(* CODESYS project PLC 1 Simulatie Ladder StructuredTekst IOStructures 2V0.project
   Title: Simulatie Sorteer Station
   Author: Rene Potters/Gerard Harkema
   Version: 0.1.0
   Description: Simulatie voor opstelling Sorteer Station.
   Company: Avans

Project tree, tasks and I/O mapping:
  Device : EHV-CPU1025, Hitachi-IES, order no. EHV-CPU1025, version 3.5.4.11
      settings: IP Address = '192.168.1.31'
    application ApplicationLadder
      libraries: VisuDialogs, * (System); Standard, 3.5.14.0 (System); Util, 3.5.14.0 (System)
      task MainTask (cyclic, interval t#20ms, priority 1) calls BedieningPrg, HoofdPrg, MagazijnPrg, OverzetterPrg, SorterenPrg, SignaleringPrg
      task Simulatie (cyclic, interval 50 ms, priority 1) calls MagazijnSim [Afhandeling Magazijn], OverzetterSim [Afhandeling Overzetter], SorterenSim [Afhandeling Sorteren]
    application ApplicationSt
      libraries: Standard, * (System); Util, * (System); VisuDialogs, 3.5.12.0 (System)
      task MainTask (cyclic, interval t#20ms, priority 1) calls Main
      task Simulatie (cyclic, interval t#20ms, priority 1) calls MagazijnSim, OverzetterSim, SorterenSim
    application MagazijnTest
      libraries: Standard, * (System); Util, * (System); VisuDialogs, 3.5.12.0 (System)
      task MainTask (cyclic, interval t#20ms, priority 1) calls MagazijnTest
      task Simulatie (cyclic, interval t#20ms, priority 1) calls MagazijnSim
    application OverzetterTest
      libraries: Standard, * (System); Util, * (System); VisuDialogs, 3.5.12.0 (System)
      task MainTask (cyclic, interval t#20ms, priority 1) calls OverzetterTest
      task Simulatie (cyclic, interval t#20ms, priority 1) calls OverzetterSim
    application SorteerTest
      libraries: Standard, * (System); Util, * (System); VisuDialogs, 3.5.12.0 (System)
      task MainTask (cyclic, interval t#20ms, priority 1) calls SorteerTest
      task Simulatie (cyclic, interval 20 ms, priority 1) calls SorterenSim
    application UitvoerGootTest
      libraries: Standard, * (System); Util, * (System); VisuDialogs, 3.5.12.0 (System)
      task MainTask (cyclic, interval t#20ms, priority 1) calls UitvoerGootTest
      task Simulatie (cyclic, interval t#20ms, priority 1) calls SorterenSim
    Basic : Basic, Hitachi-IES, version 3.4.4.0
      <Empty>
      <Empty>
      <Empty>
      <Empty>
      <Empty>
      <Empty>
      <Empty>
      <Empty>
      <Empty>
      <Empty>
      <Empty>
  Simulatie/
    program MagazijnSim [ST]
    program SorterenSim [ST]
    global variables SIM
    program OverzetterSim [ST]
    data type OverzetterDUT
    data type SorterenDUT
    data type MagazijnDUT
    function block SorterenGootSim [ST]
  Programma Ladder/
    program MagazijnPrg [SFC]
    program HoofdPrg [SFC]
    program OverzetterPrg [SFC]
    program SorterenPrg [SFC]
    program BedieningPrg [LD]
    program SignaleringPrg [LD]
  text list GlobalTextList
  Programma Structured Text/
    function block OverzetterClass [ST]: initialize, cycle, isError, isKlaar, reset, start, noodstop
    function block SorteerGootClass [ST]: initialize, cycle, isError, isKlaar, start, reset, noodstop, isGootVol, productTellerReset
    function block MagazijnClass [ST]: initialize, cycle, start, isMagazijnLeeg, isError, reset, isKlaar, noodstop
    program Main [ST]
    function block SorteerStationClass [ST]: initialize, cycle
    TestProgramms/
      program MagazijnTest [ST]
      program OverzetterTest [ST]
      program SorteerTest [ST]
      program UitvoerGootTest [ST]
    States/
      data type magazijnStates
      data type overzetterStates
      data type sorteerStationStates
      data type sorteerStates
      data type uitvoerGootStates
    function block MeetstationClass [ST]: initialize, getProductType
    data type productType
    function block UitvoerGootClass [ST]: cycle, initialize, isError, noodstop, reset, gaUit, gaIn, isUit, isIn
    Structures/
      data type uitvoerGootIO
      data type sorteerGootIO
      data type meetstationIO
      data type magazijnIO
      data type overzetterIO
      data type sorteerStationIO
      data type hmiIO
  global variables GVL
  Visualisaties/
    visualisation SorteerStationHMI
    visualisation BekerMagazijnHMI
    visualisation OverzetterHMI
    visualisation SorterenHMI
*)

// Simulatie/OverzetterDUT
{attribute 'qualified_only'}
{attribute 'strict'}
TYPE OverzetterDUT :
(
	INHETMIDDEN, NAARRECHTS, ISRECHTS, NAARLINKS, ISLINKS, GEVALLEN
);
END_TYPE

// Simulatie/SorterenDUT
{attribute 'qualified_only'}
{attribute 'strict'}
TYPE SorterenDUT :
(
	VOLGENDEBLOK, OPDEBAND, VOORSTOPPER, NAARGOOT1, INGOOT1, NAARGOOT2, INGOOT2, NAARGOOT3, INGOOT3, GEREED, VOL
);
END_TYPE

// Simulatie/MagazijnDUT
{attribute 'qualified_only'}
{attribute 'strict'}
TYPE MagazijnDUT :
(
	INGETROKKEN, INTREKKEN, UITGESTOTEN, UITSTOTEN, LEEG
);
END_TYPE

// Programma Structured Text/States/magazijnStates
// Datum : 17 december 2020, Auteur: Gerard Harkema
{attribute 'qualified_only'}
{attribute 'strict'}
TYPE magazijnStates :
(
	idle := 0,
	in,
	travel_out,
	out,
	travel_in,
	error
);
END_TYPE

// Programma Structured Text/States/overzetterStates
// Datum : 17 december 2020, Auteur: Gerard Harkema
{attribute 'qualified_only'}
{attribute 'strict'}
TYPE overzetterStates :
(
	idle := 0,
	is_links,
	vaccuum_aanzetten,
	ga_naar_rechts,
	is_rechts,
	vaccuum_lossen,
	ga_naar_midden,
	is_midden,
	ga_naar_links,
	error
);
END_TYPE

// Programma Structured Text/States/sorteerStationStates
// Datum : 17 december 2020, Auteur: Gerard Harkema
{attribute 'qualified_only'}
{attribute 'strict'}
TYPE sorteerStationStates :
(
	idle := 0,
	wacht_op_klaar,
	wacht_enable,
	product_uitgifte,
	product_overzetten,
	product_sorteren,
	service,
	error
);
END_TYPE

// Programma Structured Text/productType
// Datum : 17 december 2020, Auteur: Gerard Harkema
{attribute 'qualified_only'}
{attribute 'strict'}
TYPE productType :
(
	onbekend := 0,
	metaal_blank,
	metaal_zwart,
	kunstof_rood,
	kunstof_zwart
);
END_TYPE

// Programma Structured Text/States/sorteerStates
// Datum : 17 december 2020, Auteur: Gerard Harkema
{attribute 'qualified_only'}
{attribute 'strict'}
TYPE sorteerStates :
(
	idle := 0,
	wacht_op_start,
	stopper_uit,
	meten,
	uitvoer_goot_uit,
	transporteren_naar_goot,
	uitvoer_goot_in,
	goot_vol,
	error,
	reset_error
);
END_TYPE

// Programma Structured Text/States/uitvoerGootStates
// Datum : 17 december 2020, Auteur: Gerard Harkema
{attribute 'qualified_only'}
{attribute 'strict'}
TYPE uitvoerGootStates :
(
	idle := 0,
	is_in,
	ga_in,
	is_uit,
	ga_uit,
	error
);
END_TYPE

// Programma Structured Text/Structures/uitvoerGootIO
// Datum : 17 december 2020, Auteur: Gerard Harkema
TYPE uitvoerGootIO :
STRUCT
	//Pusher uitvoergoo is in
	Ix_UitvoerGootIsIn 		: REFERENCE TO BOOL;
	//Pusher uitvoergoot is uit
	Ix_UitvoerGootIsUit 	: REFERENCE TO BOOL;
	//Pusher goot uit
	Qx_UitvoerGootUit 		: REFERENCE TO BOOL;
END_STRUCT
END_TYPE

// Programma Structured Text/Structures/sorteerGootIO
// Datum : 17 december 2020, Auteur: Gerard Harkema
TYPE sorteerGootIO :
STRUCT
		//Product is naar een van de goten gegaan
	Ix_BekerInGoot 			:REFERENCE TO BOOL;
	//Pusher uitvoergoot 1 is in
	Ix_UitvoerGoot1IsIn 	:REFERENCE TO BOOL;
	//Pusher uitvoergoot 2 is in
	Ix_UitvoerGoot2IsIn 	:REFERENCE TO BOOL;
	//Beker afvoeren is bezig
	Ix_StationAfvoerVrij 	:REFERENCE TO BOOL;
	//Pusher uitvoergoot 1 is uit
	Ix_UitvoerGoot1IsUit 	:REFERENCE TO BOOL;
	//Pusher uitvoergoot 2 is uit
	Ix_UitvoerGoot2IsUit 	:REFERENCE TO BOOL;

	//Transportband aan
	Qx_MotorAfvoerAan 		:REFERENCE TO BOOL;
	//Pusher goot 1 uit
	Qx_UitvoerGoot1Uit 		:REFERENCE TO BOOL;
	//Pusher goot 2 uit
	Qx_UitvoerGoot2Uit 		:REFERENCE TO BOOL;
	//Beker stoppen op band voor detectie
	Qx_StopperUit 			:REFERENCE TO BOOL;
	//Uitsorteren is bezet
	Qx_StationBezet 		:REFERENCE TO BOOL;
	
	uitvoerGoot1			:uitvoerGootIO;
	uitvoerGoot2			:uitvoerGootIO;
	meetstation				:meetstationIO;

 
END_STRUCT
END_TYPE

// Programma Structured Text/Structures/meetstationIO
// Datum : 17 december 2020, Auteur: Gerard Harkema
TYPE meetstationIO :
STRUCT
	//Beker aanwezig op detectiepositie
	Ix_BekerAanwezig :REFERENCE TO BOOL;
	//Beker is van aluminium
	Ix_BekerMetaal :REFERENCE TO BOOL;
	//Beker reflecteert en is dus niet zwart
	Ix_BekerReflecteerd :REFERENCE TO BOOL;
END_STRUCT
END_TYPE

// Programma Structured Text/Structures/magazijnIO
// Datum : 17 december 2020, Auteur: Gerard Harkema
TYPE magazijnIO :
STRUCT
	// Bekers magazijn zijn op
	Ix_MagazijnLeeg				: REFERENCE TO BOOL;
	// Beker is uit dekselmagazijn gestoten
	Ix_UitstoterBekerIn			: REFERENCE TO BOOL;
	// Uitstoter Beker haalt nieuwe beker op
	Ix_UitstoterBekerUit		: REFERENCE TO BOOL;
	// Beker uit magazijn stoten
	Qx_BekerUitstoten			: REFERENCE TO BOOL;

	//Perslucht is aanwezig
	Ix_PersluchtAanwezig 		: REFERENCE TO BOOL;

END_STRUCT
END_TYPE

// Programma Structured Text/Structures/overzetterIO
// Datum : 17 december 2020, Auteur: Gerard Harkema
TYPE overzetterIO :
STRUCT
	//Werkstuk door overzetter opgepakt
	Ix_VacuumAanwezig 		:REFERENCE TO BOOL;
	//Overzetter haalt beker op(linker pos.)
	Ix_OverzetterIsLinks 	:REFERENCE TO BOOL;
	//Overzetter plaatst beker op sorteerpositie
	Ix_OverzetterIsRechts 	:REFERENCE TO BOOL;
	//Beker aanwezig op detectiepositie
	
		//Beker oppakken
	Qx_VacuumAan 			:REFERENCE TO BOOL;
	//Beker loslaten
	Qx_BekerLossen 			:REFERENCE TO BOOL;
	//Overzetter naar bekermagazijn
	Qx_OverzetterLinks 		:REFERENCE TO BOOL;
	//Overzetter naar sorteerpositie
	Qx_OverzetterRechts 	:REFERENCE TO BOOL;

END_STRUCT
END_TYPE

// Programma Structured Text/Structures/sorteerStationIO
// Datum : 17 december 2020, Auteur: Gerard Harkema
TYPE sorteerStationIO :
STRUCT
	magazijn		: magazijnIO;
	overzetter		: overzetterIO;
	sorteerGoot		: sorteerGootIO;
	hmi				: hmiIO;
END_STRUCT
END_TYPE

// Programma Structured Text/Structures/hmiIO
// Datum : 17 december 2020, Auteur: Gerard Harkema
TYPE hmiIO :
STRUCT
	// Indrukken resetknop 
	Ix_Resetknop			: REFERENCE TO BOOL;
	// Keuzeknop staat op hand
	Ix_Hand					: REFERENCE TO BOOL;
	// Keuzeknop staat op auto
	Ix_Auto					: REFERENCE TO BOOL;
	// Indrukken noodstop
	Ix_Noodstop				: REFERENCE TO BOOL;
	// Bekers magazijn zijn op

	// Indrukken startknop
	Ix_Stopknop				: REFERENCE TO BOOL;
	// Indrukken stopknop
	Ix_Startknop			: REFERENCE TO BOOL;	
	//Perslucht is aanwezig

	// Visualisatie invisible Gele vlak
	Qx_GeleLamp				: REFERENCE TO BOOL;
	// Visualisatie invisible groene vlak
	Qx_GroeneLamp			: REFERENCE TO BOOL;
	// Visualisatie invisible rode vlak
	Qx_RodeLamp				: REFERENCE TO BOOL;

END_STRUCT
END_TYPE

// Simulatie/SIM
{attribute 'qualified_only'}
VAR_GLOBAL
	// Rotatie van de overzetter
	Vx_OvzRotate: INT := 0;
	// Visualisatie invisible blok
	Vx_OvzBlokLinks: BOOL := FALSE;
	// Visualisatie invisible blok
	Vx_OvzBlokOverzetter: BOOL := FALSE;
	// Visualisatie invisible blok
	Vx_OvzBlokRechts: BOOL := FALSE;
	// Visualisatie invisible blok
	Vx_OvzBlokGevallen: BOOL := FALSE;	
	// Magazijn opnieuw vullen (simulatie)
	Ix_MagazijnVullen 	: BOOL;
	// Goten legen (symulatie)
	Ix_GotenLegen	  	: BOOL;
	
	
	
	
	
	
	
	
	
	
	
	
	
	
	
	
	
	
	
	
	
	
	
	
	
	
	
	
	
	
	
	
	
	
	
	
	
	
	
	
	
	
	
	
	
	
	
	
	// Simulatie visualisatie 
	Vw_Rotate45: INT := 45;
	// Visualisatie X positie van de uitstoter
	Vw_MagUitstoterBekerX: INT := 30;
	// Visualisatie invisible blok uitgestoten
	Vx_MagBlokUit: BOOL := TRUE;
	// Visualisatie invisible blok 1
	Vx_MagBlok1: BOOL := TRUE;
	// Visualisatie invisible blok 2
	Vx_MagBlok2: BOOL := TRUE;
	// Visualisatie invisible blok 3
	Vx_MagBlok3: BOOL := TRUE;
	// Visualisatie invisible blok 4
	Vx_MagBlok4: BOOL := TRUE;
	// Visualisatie invisible blokken
	Vx_MagBlok: ARRAY[1..8] OF BOOL;
	// Aantal blokken in het magazijn
	Vw_MagBlokAantal: INT := 4;
	// Simulatie onthoudt dat een blok maar 1x wordt uitgestoten
	Vw_MagBlok1X: INT := 0;
	// Ligt er een blok op band
	Vw_SorBlokBand: BOOL := FALSE;
	// Rotatie van de stopper
	Vw_SorStopperRotate: INT := 0;
	// Rotatie van de stopper goot 1
	Vw_SorGoot1Rotate: INT := 0;
	// Rotatie van de stopper goot 2
	Vw_SorGoot2Rotate: INT := 0;
	// Kleur van de blok op betreffende positie
	Vw_SorKleurBand: DWORD := 0;
	// Bewegen van de blok over de band
	Vi_SorBlokBandX: INT := 0;
	// Bewegen van de blok over de band
	Vi_SorBlokBandY: INT := 0;
	// Simulatie error. Inverse logica.
	Vx_MagLuchtDrukError: BOOL := TRUE;
	// Simulatie error. Inverse logica.
	Vx_MagIsInError: BOOL := TRUE;
	// Simulatie error. Inverse logica.
	Vx_MagIsUitError: BOOL := TRUE;
	// Simulatie error. Inverse logica.
	Vx_OvzLuchtDrukError: BOOL := TRUE;
	// Simulatie error. Inverse logica.
	Vx_OvzIsLinksError: BOOL := TRUE;
	// Simulatie error. Inverse logica.
	Vx_OvzIsRechtsError: BOOL := TRUE;
	// Simulatie error. Inverse logica.
	Vx_OvzVacuumError: BOOL := TRUE;
	// Simulatie error. Inverse logica.
	Vx_SorMotorAfvoerError: BOOL := TRUE;
	// Simulatie error. Inverse logica.
	Vx_SorGoot1InError: BOOL := TRUE;
	// Simulatie error. Inverse logica.
	Vx_SorGoot1UitError: BOOL := TRUE;
	// Simulatie error. Inverse logica.
	Vx_SorInGootError: BOOL := TRUE;
	// Ligt er een blok op de betreffende positie
	Vx_SorBlokGoot: ARRAY [1..3,1..6] OF BOOL;
	// Kleur van de blok op betreffende positie
	Vw_SorKleurGoot: ARRAY [1..3,1..6] OF DWORD;
END_VAR

// GVL
VAR_GLOBAL
	// Indrukken resetknop 
	Ix_Resetknop: BOOL;
	// Keuzeknop staat op hand
	Ix_Hand: BOOL;
	// Keuzeknop staat op auto
	Ix_Auto: BOOL;
	// Indrukken noodstop
	Ix_Noodstop: BOOL;
	// Bekers magazijn zijn op
	Ix_MagazijnLeeg: BOOL;
	// Beker is uit dekselmagazijn gestoten
	Ix_UitstoterBekerIn: BOOL;
	// Uitstoter Beker haalt nieuwe beker op
	Ix_UitstoterBekerUit: BOOL;
	// Indrukken startknop
	Ix_Stopknop: BOOL := TRUE;
	// Indrukken stopknop
	Ix_Startknop: BOOL;	
	//Perslucht is aanwezig
	Ix_PersluchtAanwezig :BOOL;
	//Werkstuk door overzetter opgepakt
	Ix_VacuumAanwezig :BOOL;
	//Overzetter haalt beker op(linker pos.)
	Ix_OverzetterIsLinks :BOOL;
	//Overzetter plaatst beker op sorteerpositie
	Ix_OverzetterIsRechts :BOOL;
	//Beker aanwezig op detectiepositie
	Ix_BekerAanwezig :BOOL;
	//Beker is van aluminium
	Ix_BekerMetaal :BOOL;
	//Beker reflecteert en is dus niet zwart
	Ix_BekerReflecteerd :BOOL;
	//Product is naar een van de goten gegaan
	Ix_BekerInGoot :BOOL;
	//Pusher uitvoergoot 1 is in
	Ix_UitvoerGoot1IsIn :BOOL;
	//Pusher uitvoergoot 2 is in
	Ix_UitvoerGoot2IsIn :BOOL;
	//Beker afvoeren is bezig
	Ix_StationAfvoerVrij :BOOL;
	//Pusher uitvoergoot 1 is uit
	Ix_UitvoerGoot1IsUit :BOOL;
	//Pusher uitvoergoot 2 is uit
	Ix_UitvoerGoot2IsUit :BOOL;
	// Beker uit magazijn stoten
	Qx_BekerUitstoten: BOOL;	
	//Beker oppakken
	Qx_VacuumAan :BOOL;
	//Beker loslaten
	Qx_BekerLossen :BOOL;
	//Overzetter naar bekermagazijn
	Qx_OverzetterLinks :BOOL;
	//Overzetter naar sorteerpositie
	Qx_OverzetterRechts :BOOL;
	//Transportband aan
	Qx_MotorAfvoerAan :BOOL;
	//Pusher goot 1 uit
	Qx_UitvoerGoot1Uit :BOOL;
	//Pusher goot 2 uit
	Qx_UitvoerGoot2Uit :BOOL;
	//Beker stoppen op band voor detectie
	Qx_StopperUit :BOOL;
	//Uitsorteren is bezet
	Qx_StationBezet :BOOL;
	// Visualisatie invisible Gele vlak
	Qx_GeleLamp: BOOL;
	// Visualisatie invisible groene vlak
	Qx_GroeneLamp: BOOL;
	// Visualisatie invisible rode vlak
	Qx_RodeLamp: BOOL;
	
END_VAR

// Programma Ladder/BedieningPrg
PROGRAM BedieningPrg
VAR
END_VAR

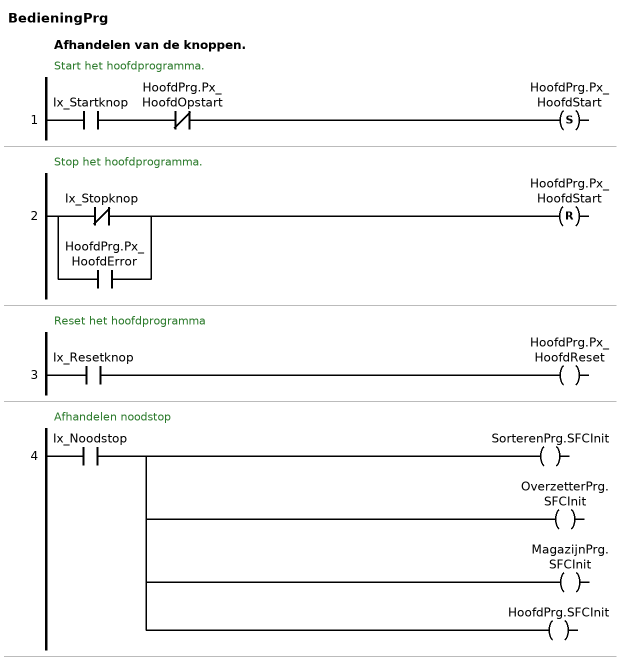
// NETWORK 1: Afhandelen van de knoppen.
// Start het hoofdprogramma.
HoofdPrg.Px_HoofdStart S= Ix_Startknop AND NOT HoofdPrg.Px_HoofdOpstart;

// NETWORK 2
// Stop het hoofdprogramma.
HoofdPrg.Px_HoofdStart R= NOT Ix_Stopknop OR HoofdPrg.Px_HoofdError;

// NETWORK 3
// Reset het hoofdprogramma
HoofdPrg.Px_HoofdReset := Ix_Resetknop;

// NETWORK 4
// Afhandelen noodstop
SorterenPrg.SFCInit := Ix_Noodstop;
OverzetterPrg.SFCInit := Ix_Noodstop;
MagazijnPrg.SFCInit := Ix_Noodstop;
HoofdPrg.SFCInit := Ix_Noodstop;

END_PROGRAM

// Programma Ladder/HoofdPrg
PROGRAM HoofdPrg
VAR_INPUT
	// Reset het programma
	Px_HoofdReset: BOOL;
	// Start het programma
	Px_HoofdStart: BOOL;
	// Reset de SFC bv Noodstop
	SFCInit: BOOL;
END_VAR
VAR_OUTPUT
	// Er is een error op getreden
	Px_HoofdError: BOOL;
	// Commando is uitgevoerd
	Px_HoofdGereed: BOOL;
	// Programma is bezig
	Px_HoofdBezig: BOOL;
	// Programma is aan het opstarten
	Px_HoofdOpstart: BOOL;
END_VAR

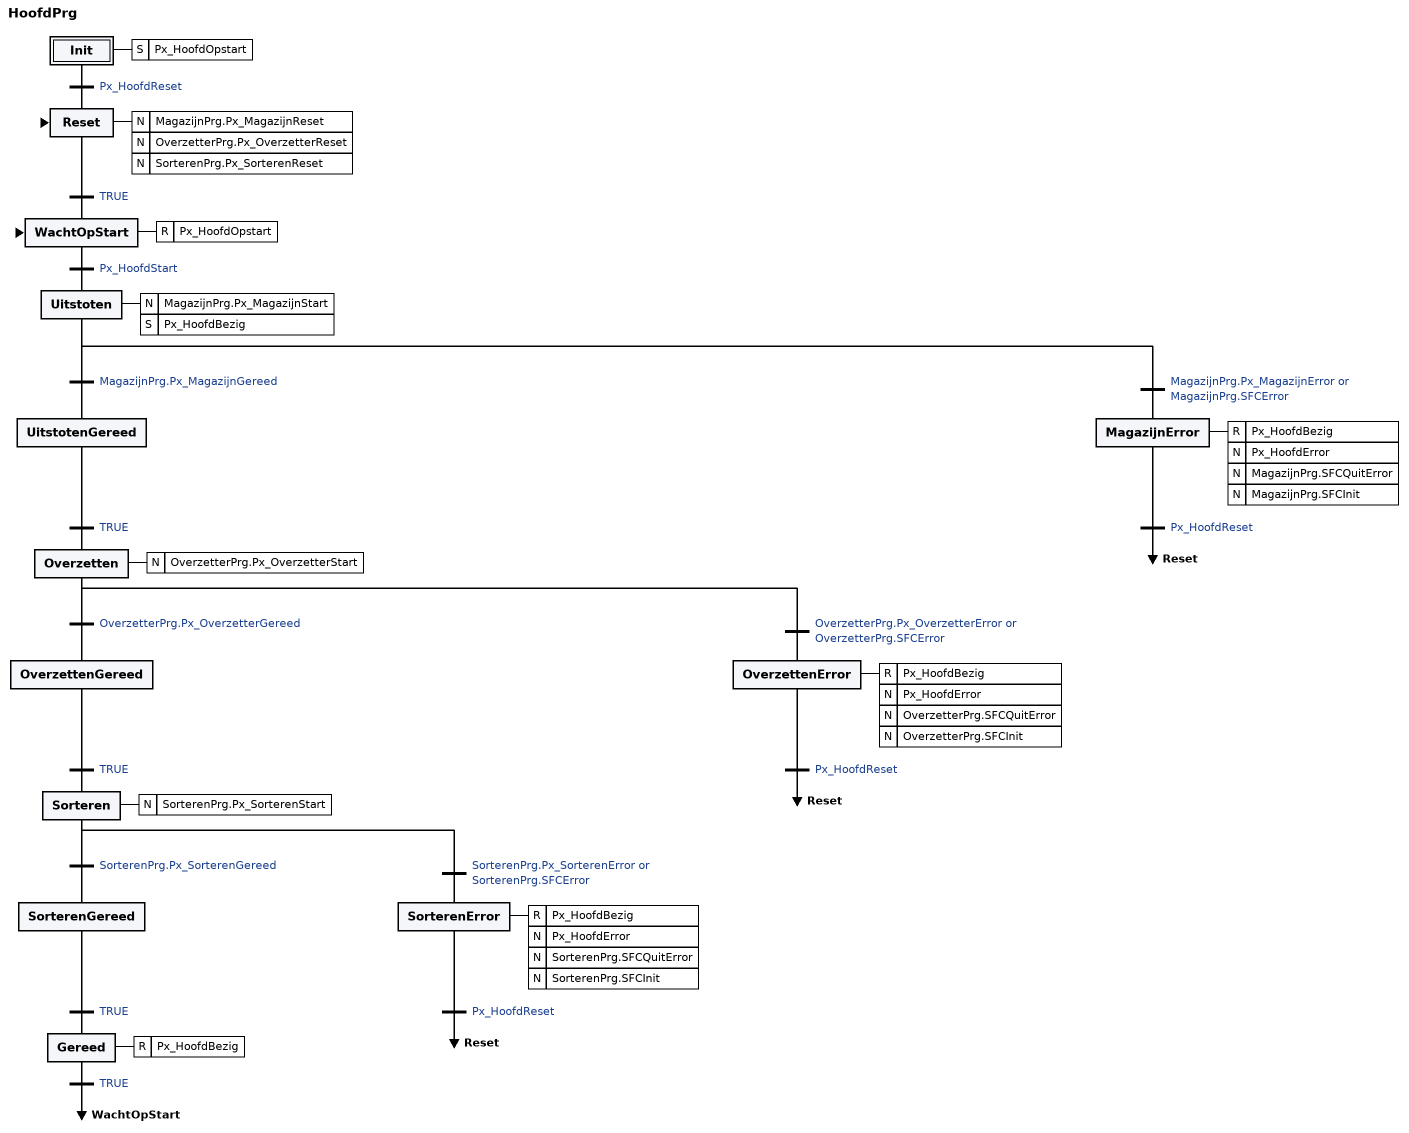
INITIAL_STEP Init:
    Px_HoofdOpstart(S);
END_STEP
TRANSITION FROM Init TO Reset
    := Px_HoofdReset;
END_TRANSITION
STEP Reset:
    MagazijnPrg.Px_MagazijnReset(N);
    OverzetterPrg.Px_OverzetterReset(N);
    SorterenPrg.Px_SorterenReset(N);
END_STEP
TRANSITION FROM Reset TO WachtOpStart
    := TRUE;
END_TRANSITION
STEP WachtOpStart:
    Px_HoofdOpstart(R);
END_STEP
TRANSITION FROM WachtOpStart TO Uitstoten
    := Px_HoofdStart;
END_TRANSITION
STEP Uitstoten:  // max time T#30S
    MagazijnPrg.Px_MagazijnStart(N);
    Px_HoofdBezig(S);
END_STEP
TRANSITION FROM Uitstoten TO UitstotenGereed
    := MagazijnPrg.Px_MagazijnGereed;
END_TRANSITION
STEP UitstotenGereed:
END_STEP
TRANSITION FROM UitstotenGereed TO Overzetten
    := TRUE;
END_TRANSITION
TRANSITION FROM Uitstoten TO MagazijnError
    := MagazijnPrg.Px_MagazijnError or MagazijnPrg.SFCError;
END_TRANSITION
STEP MagazijnError:
    Px_HoofdBezig(R);
    Px_HoofdError(N);
    MagazijnPrg.SFCQuitError(N);
    MagazijnPrg.SFCInit(N);
END_STEP
TRANSITION FROM MagazijnError TO Reset
    := Px_HoofdReset;
END_TRANSITION
STEP Overzetten:
    OverzetterPrg.Px_OverzetterStart(N);
END_STEP
TRANSITION FROM Overzetten TO OverzettenGereed
    := OverzetterPrg.Px_OverzetterGereed;
END_TRANSITION
STEP OverzettenGereed:
END_STEP
TRANSITION FROM OverzettenGereed TO Sorteren
    := TRUE;
END_TRANSITION
TRANSITION FROM Overzetten TO OverzettenError
    := OverzetterPrg.Px_OverzetterError or OverzetterPrg.SFCError;
END_TRANSITION
STEP OverzettenError:
    Px_HoofdBezig(R);
    Px_HoofdError(N);
    OverzetterPrg.SFCQuitError(N);
    OverzetterPrg.SFCInit(N);
END_STEP
TRANSITION FROM OverzettenError TO Reset
    := Px_HoofdReset;
END_TRANSITION
STEP Sorteren:
    SorterenPrg.Px_SorterenStart(N);
END_STEP
TRANSITION FROM Sorteren TO SorterenGereed
    := SorterenPrg.Px_SorterenGereed;
END_TRANSITION
STEP SorterenGereed:
END_STEP
TRANSITION FROM SorterenGereed TO Gereed
    := TRUE;
END_TRANSITION
TRANSITION FROM Sorteren TO SorterenError
    := SorterenPrg.Px_SorterenError or SorterenPrg.SFCError;
END_TRANSITION
STEP SorterenError:
    Px_HoofdBezig(R);
    Px_HoofdError(N);
    SorterenPrg.SFCQuitError(N);
    SorterenPrg.SFCInit(N);
END_STEP
TRANSITION FROM SorterenError TO Reset
    := Px_HoofdReset;
END_TRANSITION
STEP Gereed:
    Px_HoofdBezig(R);
END_STEP
TRANSITION FROM Gereed TO WachtOpStart
    := TRUE;
END_TRANSITION

END_PROGRAM

// Programma Ladder/SorterenPrg
PROGRAM SorterenPrg
VAR_INPUT
	// Reset de sorteren na start of error
	Px_SorterenReset: BOOL;
	// Start het sorteren
	Px_SorterenStart: BOOL;
	
	// Reset de SFC bv Noodstop
	SFCInit: BOOL;
	// Enable runtime limit checks
	SFCEnableLimit: BOOL := TRUE;	
	// Reset runtime error
	SFCQuitError : BOOL;	
END_VAR
VAR_OUTPUT
	// Sorteren heeft een error
	Px_SorterenError: BOOL;
	// Sorteren heeft een opdracht uitgevoerd
	Px_SorterenGereed: BOOL;
	// Sorteren is bezig
	Px_SorterenBezig: BOOL;
	// Runtime limit is opgetreden
	SFCError: BOOL;		
END_VAR

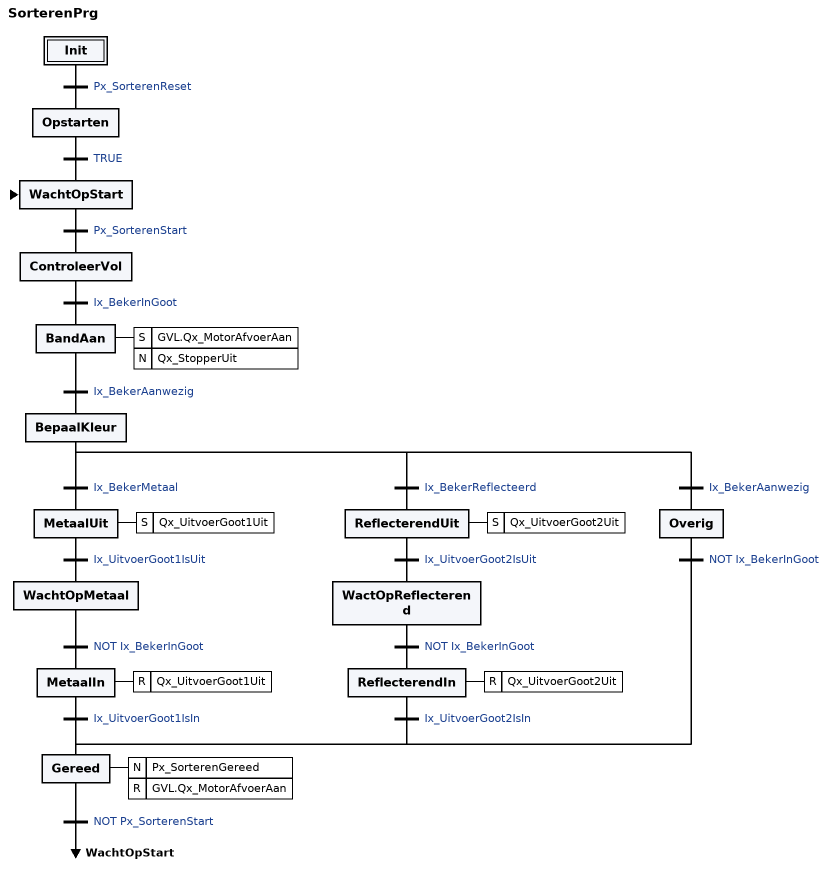
INITIAL_STEP Init:
END_STEP
TRANSITION FROM Init TO Opstarten
    := Px_SorterenReset;
END_TRANSITION
STEP Opstarten:
END_STEP
TRANSITION FROM Opstarten TO WachtOpStart
    := TRUE;
END_TRANSITION
STEP WachtOpStart:
END_STEP
TRANSITION FROM WachtOpStart TO ControleerVol
    := Px_SorterenStart;
END_TRANSITION
STEP ControleerVol:  // max time T#1S
END_STEP
TRANSITION FROM ControleerVol TO BandAan
    := Ix_BekerInGoot;
END_TRANSITION
STEP BandAan:
    GVL.Qx_MotorAfvoerAan(S);
    Qx_StopperUit(N);
END_STEP
TRANSITION FROM BandAan TO BepaalKleur
    := Ix_BekerAanwezig;
END_TRANSITION
STEP BepaalKleur:  // max time T#15S
END_STEP
TRANSITION FROM BepaalKleur TO MetaalUit
    := Ix_BekerMetaal;
END_TRANSITION
STEP MetaalUit:  // max time T#15S
    Qx_UitvoerGoot1Uit(S);
END_STEP
TRANSITION FROM MetaalUit TO WachtOpMetaal
    := Ix_UitvoerGoot1IsUit;
END_TRANSITION
STEP WachtOpMetaal:  // max time T#15S
END_STEP
TRANSITION FROM WachtOpMetaal TO MetaalIn
    := NOT Ix_BekerInGoot;
END_TRANSITION
STEP MetaalIn:  // max time T#15S
    Qx_UitvoerGoot1Uit(R);
END_STEP
TRANSITION FROM MetaalIn TO Gereed
    := Ix_UitvoerGoot1IsIn;
END_TRANSITION
TRANSITION FROM BepaalKleur TO ReflecterendUit
    := Ix_BekerReflecteerd;
END_TRANSITION
STEP ReflecterendUit:  // max time T#15S
    Qx_UitvoerGoot2Uit(S);
END_STEP
TRANSITION FROM ReflecterendUit TO WactOpReflecterend
    := Ix_UitvoerGoot2IsUit;
END_TRANSITION
STEP WactOpReflecterend:  // max time T#15S
END_STEP
TRANSITION FROM WactOpReflecterend TO ReflecterendIn
    := NOT Ix_BekerInGoot;
END_TRANSITION
STEP ReflecterendIn:  // max time T#15S
    Qx_UitvoerGoot2Uit(R);
END_STEP
TRANSITION FROM ReflecterendIn TO Gereed
    := Ix_UitvoerGoot2IsIn;
END_TRANSITION
TRANSITION FROM BepaalKleur TO Overig
    := Ix_BekerAanwezig;
END_TRANSITION
STEP Overig:  // max time T#15S
END_STEP
TRANSITION FROM Overig TO Gereed
    := NOT Ix_BekerInGoot;
END_TRANSITION
STEP Gereed:
    Px_SorterenGereed(N);
    GVL.Qx_MotorAfvoerAan(R);
END_STEP
TRANSITION FROM Gereed TO WachtOpStart
    := NOT Px_SorterenStart;
END_TRANSITION

END_PROGRAM

// Programma Ladder/OverzetterPrg
PROGRAM OverzetterPrg
VAR_INPUT
	// Reset de overzetter na start of error
	Px_OverzetterReset: BOOL;
	// Start de overzetter
	Px_OverzetterStart: BOOL;
	
	// Reset de SFC bv Noodstop
	SFCInit: BOOL;
	// Enable runtime limit checks
	SFCEnableLimit: BOOL := TRUE;	
	// Reset runtime error
	SFCQuitError : BOOL;	
END_VAR
VAR_OUTPUT
	// Overzetter heeft een error
	Px_OverzetterError: BOOL;
	// Overzetter heeft opdracht uitgevoerd
	Px_OverzetterGereed: BOOL;
	// Overzetter is bezig
	Px_OverzetterBezig: BOOL;
	// Runtime limit is opgetreden
	SFCError: BOOL;		
END_VAR
VAR
	// Tijdsvertraging voor sommige stappen
	Mx_Delay: BOOL;
END_VAR

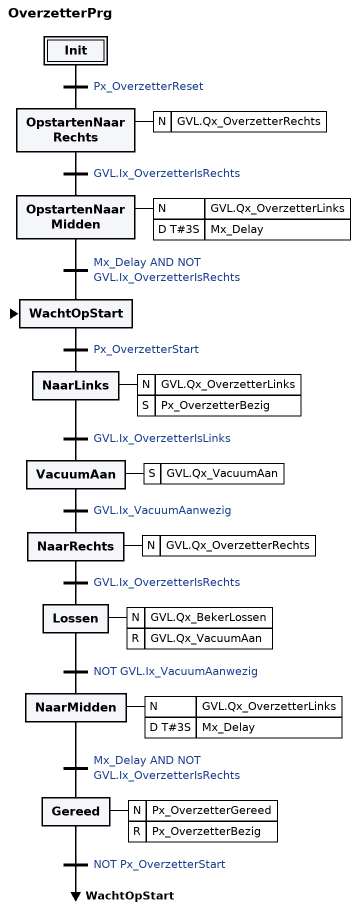
INITIAL_STEP Init:
END_STEP
TRANSITION FROM Init TO OpstartenNaarRechts
    := Px_OverzetterReset;
END_TRANSITION
STEP OpstartenNaarRechts:  // max time T#15S
    GVL.Qx_OverzetterRechts(N);
END_STEP
TRANSITION FROM OpstartenNaarRechts TO OpstartenNaarMidden
    := GVL.Ix_OverzetterIsRechts;
END_TRANSITION
STEP OpstartenNaarMidden:  // max time T#10S
    GVL.Qx_OverzetterLinks(N);
    Mx_Delay(D, T#3S);
END_STEP
TRANSITION FROM OpstartenNaarMidden TO WachtOpStart
    := Mx_Delay AND NOT GVL.Ix_OverzetterIsRechts;
END_TRANSITION
STEP WachtOpStart:
END_STEP
TRANSITION FROM WachtOpStart TO NaarLinks
    := Px_OverzetterStart;
END_TRANSITION
STEP NaarLinks:  // max time T#15S
    GVL.Qx_OverzetterLinks(N);
    Px_OverzetterBezig(S);
END_STEP
TRANSITION FROM NaarLinks TO VacuumAan
    := GVL.Ix_OverzetterIsLinks;
END_TRANSITION
STEP VacuumAan:  // max time T#15S
    GVL.Qx_VacuumAan(S);
END_STEP
TRANSITION FROM VacuumAan TO NaarRechts
    := GVL.Ix_VacuumAanwezig;
END_TRANSITION
STEP NaarRechts:  // max time T#15S
    GVL.Qx_OverzetterRechts(N);
END_STEP
TRANSITION FROM NaarRechts TO Lossen
    := GVL.Ix_OverzetterIsRechts;
END_TRANSITION
STEP Lossen:  // max time T#15S
    GVL.Qx_BekerLossen(N);
    GVL.Qx_VacuumAan(R);
END_STEP
TRANSITION FROM Lossen TO NaarMidden
    := NOT GVL.Ix_VacuumAanwezig;
END_TRANSITION
STEP NaarMidden:  // max time T#15S
    GVL.Qx_OverzetterLinks(N);
    Mx_Delay(D, T#3S);
END_STEP
TRANSITION FROM NaarMidden TO Gereed
    := Mx_Delay AND NOT GVL.Ix_OverzetterIsRechts;
END_TRANSITION
STEP Gereed:
    Px_OverzetterGereed(N);
    Px_OverzetterBezig(R);
END_STEP
TRANSITION FROM Gereed TO WachtOpStart
    := NOT Px_OverzetterStart;
END_TRANSITION

END_PROGRAM

// Programma Ladder/MagazijnPrg
PROGRAM MagazijnPrg

VAR_INPUT
	// Reset het magazijn na start of error
	Px_MagazijnReset: BOOL;
	// Start uitstoten
	Px_MagazijnStart: BOOL;

	// Reset de SFC bv Noodstop
	SFCInit: BOOL;
	// Enable runtime limit checks
	SFCEnableLimit: BOOL := TRUE;	
	// Reset runtime error
	SFCQuitError : BOOL;
END_VAR

VAR_OUTPUT
	// Er is een error opgetreden
	Px_MagazijnError: BOOL;
	// Commando is uitgevoerd
	Px_MagazijnGereed: BOOL;
	// Bezig met uitvoeren van commando
	Px_MagazijnBezig: BOOL;
	// Runtime limit is opgetreden
	SFCError: BOOL;	
END_VAR

VAR
	// Tijdsvertraging voor fouten
	Mx_Error: BOOL;
END_VAR

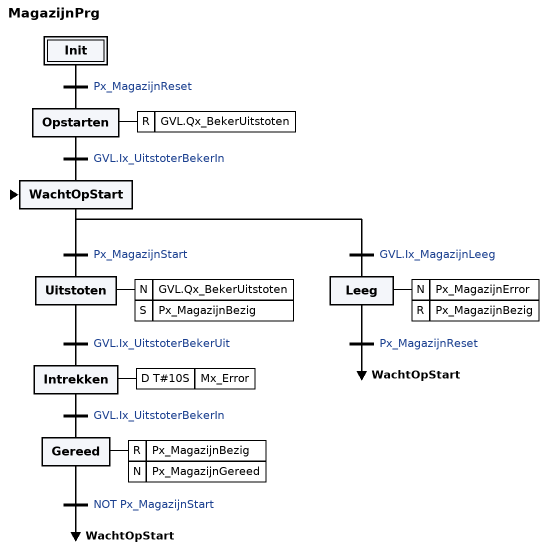
INITIAL_STEP Init:
END_STEP
TRANSITION FROM Init TO Opstarten
    := Px_MagazijnReset;
END_TRANSITION
STEP Opstarten:  // max time T#10S
    GVL.Qx_BekerUitstoten(R);
END_STEP
TRANSITION FROM Opstarten TO WachtOpStart
    := GVL.Ix_UitstoterBekerIn;
END_TRANSITION
STEP WachtOpStart:
END_STEP
TRANSITION FROM WachtOpStart TO Uitstoten
    := Px_MagazijnStart;
END_TRANSITION
STEP Uitstoten:  // max time T#10S
    GVL.Qx_BekerUitstoten(N);
    Px_MagazijnBezig(S);
END_STEP
TRANSITION FROM Uitstoten TO Intrekken
    := GVL.Ix_UitstoterBekerUit;
END_TRANSITION
STEP Intrekken:  // max time T#10S
    Mx_Error(D, T#10S);
END_STEP
TRANSITION FROM Intrekken TO Gereed
    := GVL.Ix_UitstoterBekerIn;
END_TRANSITION
STEP Gereed:
    Px_MagazijnBezig(R);
    Px_MagazijnGereed(N);
END_STEP
TRANSITION FROM Gereed TO WachtOpStart
    := NOT Px_MagazijnStart;
END_TRANSITION
TRANSITION FROM WachtOpStart TO Leeg
    := GVL.Ix_MagazijnLeeg;
END_TRANSITION
STEP Leeg:
    Px_MagazijnError(N);
    Px_MagazijnBezig(R);
END_STEP
TRANSITION FROM Leeg TO WachtOpStart
    := Px_MagazijnReset;
END_TRANSITION

END_PROGRAM

// Programma Ladder/SignaleringPrg
PROGRAM SignaleringPrg
VAR
	// Knipperen gele lamp
	Fb_GeelKnipper: Blink;
END_VAR

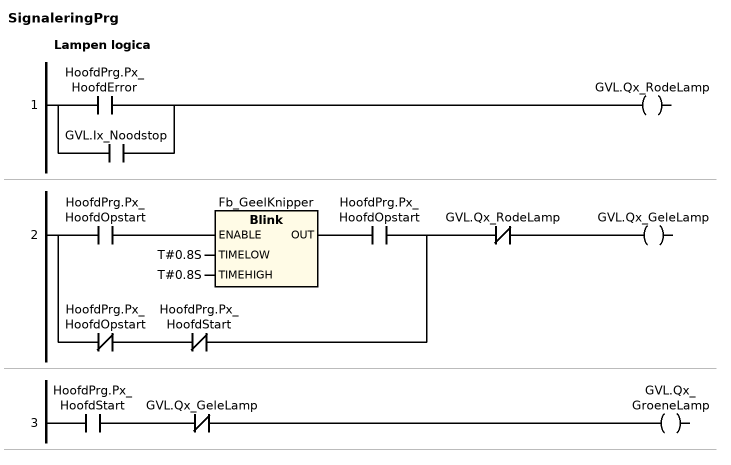
// NETWORK 1: Lampen logica
GVL.Qx_RodeLamp := HoofdPrg.Px_HoofdError OR GVL.Ix_Noodstop;

// NETWORK 2
Fb_GeelKnipper(ENABLE := HoofdPrg.Px_HoofdOpstart, TIMELOW := T#0.8S, TIMEHIGH := T#0.8S); // Blink
GVL.Qx_GeleLamp := (Fb_GeelKnipper.OUT AND HoofdPrg.Px_HoofdOpstart OR NOT HoofdPrg.Px_HoofdOpstart AND NOT HoofdPrg.Px_HoofdStart) AND NOT GVL.Qx_RodeLamp;

// NETWORK 3
GVL.Qx_GroeneLamp := HoofdPrg.Px_HoofdStart AND NOT GVL.Qx_GeleLamp;

END_PROGRAM

// Simulatie/MagazijnSim
PROGRAM MagazijnSim
VAR
	// Timer om uitstoten en intrekken te vertragen
	Fb_Pulse: BLINK;
	// Timer om intrekken te vertragen
	Fb_Trigger: F_TRIG;
	// Eerste keer om visualisatie te updaten
	Mx_FirstTime: BOOL := TRUE;
	// Afhandeling van het magazijn
	Me_MagState: MAGAZIJNDUT := MAGAZIJNDUT.INGETROKKEN;
END_VAR

//
// Common stuff.
//

IF (Mx_FirstTime) THEN
	SIM.Vw_MagBlokAantal := 8;
	SIM.Vx_MagBlokUit:= FALSE;
	
	Mx_FirstTime := FALSE;
END_IF

					
//
// Handle all pulse and trigger events.
//
Fb_Pulse(ENABLE:=TRUE,TIMELOW:=T#200MS, TIMEHIGH:=T#200MS);
Fb_Trigger(CLK:=Fb_Pulse.OUT);


//
// Only if no emergency active, start handling the simulation.
//
IF (SIM.Ix_MagazijnVullen) THEN
	Mx_FirstTime := TRUE;
	SIM.Ix_MagazijnVullen := FALSE;
	RETURN;
END_IF
	
//
// The pulse determines the speed of the cilinder to move in
// ore move out. The cilinder is only moved if the airpressure 
// is available.
//
IF (Fb_Trigger.Q AND SIM.Vx_MagLuchtDrukError) THEN
		
			
	CASE Me_MagState OF
		MAGAZIJNDUT.INGETROKKEN:
			IF (SIM.Vx_MagBlokUit) THEN
				SIM.Vw_MagBlokAantal := SIM.Vw_MagBlokAantal - 1;
			END_IF
		
			SIM.Vw_MagUitstoterBekerX := 1;
			SIM.Vw_MagBlok1X    	  := SIM.Vw_MagUitstoterBekerX;
			SIM.Vx_MagBlokUit         := FALSE;
	
			IF (Qx_BekerUitstoten) THEN
				Me_MagState := MAGAZIJNDUT.UITSTOTEN;
			END_IF

		MAGAZIJNDUT.INTREKKEN:
			SIM.Vw_MagUitstoterBekerX := SIM.Vw_MagUitstoterBekerX - 30;
			
			IF (SIM.Vw_MagUitstoterBekerX < 0) THEN 
				SIM.Vw_MagUitstoterBekerX := 0; 
			END_IF		
			
			IF (SIM.Vw_MagUitstoterBekerX = 0) THEN
				Me_MagState := MAGAZIJNDUT.INGETROKKEN;				
			END_IF		

			IF (Qx_BekerUitstoten) THEN
				Me_MagState := MAGAZIJNDUT.UITSTOTEN;
			END_IF	
	
		MAGAZIJNDUT.UITGESTOTEN:
			SIM.Vx_MagBlokUit         := SIM.Vx_MagBlok1;
						
			IF (NOT Qx_BekerUitstoten) THEN
				Me_MagState := MAGAZIJNDUT.INTREKKEN;
			END_IF	
		
		MAGAZIJNDUT.UITSTOTEN:
			SIM.Vw_MagUitstoterBekerX := SIM.Vw_MagUitstoterBekerX + 30;
			SIM.Vw_MagBlok1X    	  := SIM.Vw_MagUitstoterBekerX;			
		
			IF (SIM.Vw_MagUitstoterBekerX > 70) THEN
				Me_MagState := MAGAZIJNDUT.UITGESTOTEN;				
			END_IF		

			IF (NOT Qx_BekerUitstoten) THEN
				Me_MagState := MAGAZIJNDUT.INTREKKEN;
			END_IF	
		
	END_CASE

	GVL.Ix_UitstoterBekerIn  := (Me_MagState = MAGAZIJNDUT.INGETROKKEN) AND SIM.Vx_MagIsInError;
	GVL.Ix_UitstoterBekerUit := (Me_MagState = MAGAZIJNDUT.UITGESTOTEN) AND SIM.Vx_MagIsUitError;	
	GVL.Ix_MagazijnLeeg 	 := (SIM.Vw_MagBlokAantal <= 0) AND (Ix_UitstoterBekerIn);	
	
	SIM.Vx_MagBlok[8] := (SIM.Vw_MagBlokAantal >= 8);
	SIM.Vx_MagBlok[7] := (SIM.Vw_MagBlokAantal >= 7);
	SIM.Vx_MagBlok[6] := (SIM.Vw_MagBlokAantal >= 6);
	SIM.Vx_MagBlok[5] := (SIM.Vw_MagBlokAantal >= 5);		
	SIM.Vx_MagBlok[4] := (SIM.Vw_MagBlokAantal >= 4);
	SIM.Vx_MagBlok[3] := (SIM.Vw_MagBlokAantal >= 3);
	SIM.Vx_MagBlok[2] := (SIM.Vw_MagBlokAantal >= 2);
	SIM.Vx_MagBlok[1] := (SIM.Vw_MagBlokAantal >= 1);	
	
END_IF

END_PROGRAM

// Simulatie/OverzetterSim
PROGRAM OverzetterSim
VAR
	// Timer om overzetten te vertragen
	Fb_Pulse: BLINK;
	// Timer om overzetten te vertragen
	Fb_Trigger: F_TRIG;
	// Eerste keer om visualisatie te updaten
	Mx_FirstTime: BOOL := TRUE;
	// Afhandeling van de overzetter
	Me_OvzState: OverzetterDUT := OVERZETTERDUT.INHETMIDDEN;	
	// Afhandeling van het blokje
	Me_BlokState: OverzetterDUT := OVERZETTERDUT.INHETMIDDEN;	
	// Duurt even voor het vacuum aanwezig is
	Mi_VacuumCntr: INT := 0;	
END_VAR
VAR CONSTANT


	// Inverse logica
	INVISABLE: BOOL := TRUE;
	// Inverse logica
	VISABLE: BOOL := FALSE;

END_VAR

// Initialisatie.

IF (Mx_FirstTime) THEN
	Me_OvzState := OVERZETTERDUT.INHETMIDDEN;
	Me_BlokState := OVERZETTERDUT.ISLINKS;
	
	Mi_VacuumCntr := 0;
	SIM.Vx_OvzRotate := 0;
	Mx_FirstTime := FALSE;
END_IF

//
// Afhandelen van de pulse events. Hierdoor loopt de simulatie los van de 
// TASK tijd.
//
Fb_Pulse(ENABLE:=TRUE,TIMELOW:=T#100MS, TIMEHIGH:=T#100MS);
Fb_Trigger(CLK:=Fb_Pulse.OUT);


//
// Only if no emergency active, start handling the simulation.
//
IF (GVL.Ix_Noodstop) THEN
	Mx_FirstTime := TRUE;	
	RETURN;
END_IF
	
//
// The pulse determines the speed of the cilinder to move in
// ore move out. The cilinder is only moved if the airpressure 
// is available.
//
IF (Fb_Trigger.Q AND SIM.Vx_OvzLuchtDrukError) THEN
	
	//
	// De status van de arm wordt los afgehandeld van het blokje. De beweging
	// van de arm staat hier namelijk helemaal los van.
	//
	
	CASE Me_OvzState OF
		
		OVERZETTERDUT.INHETMIDDEN:
			// 
			// De arm is in beweging naar links of naar rechts.
			// Indien de arm in de uiterste positie is wordt er van 
			// state gewisseld. Aangezien de arm in beweging is staan
			// de eindschakelaars uit.
			//
			
			IF (GVL.Qx_OverzetterLinks) THEN
				IF (SIM.Vx_OvzRotate > -90) THEN
					GVL.Ix_OverzetterIsLinks := FALSE;	
					GVL.Ix_OverzetterIsRechts := FALSE;			
					SIM.Vx_OvzRotate := SIM.Vx_OvzRotate - 10;
				ELSE
					Me_OvzState := OVERZETTERDUT.ISLINKS;			
				END_IF	
				
			END_IF
				 
			IF (GVL.Qx_OverzetterRechts) THEN
				IF (SIM.Vx_OvzRotate < 90) THEN
					GVL.Ix_OverzetterIsLinks := FALSE;	
					GVL.Ix_OverzetterIsRechts := FALSE;				
					SIM.Vx_OvzRotate := SIM.Vx_OvzRotate + 10;
				ELSE
					Me_OvzState := OVERZETTERDUT.ISRECHTS;				
				END_IF			
			END_IF
				
		OVERZETTERDUT.ISLINKS:
		    //
			// Arm staat in een uiterste stand. Eindschakelaar is ingeschakeld.
			// Zodra de arm weer wordt bewogen verandert de state.
			//
			
			GVL.Ix_OverzetterIsLinks := TRUE AND SIM.Vx_OvzIsLinksError;	

			IF (GVL.Qx_OverzetterRechts AND NOT GVL.Qx_OverzetterLinks) THEN
				GVL.Ix_OverzetterIsLinks := FALSE;				
				Me_OvzState := OVERZETTERDUT.INHETMIDDEN;		
			END_IF
			
		OVERZETTERDUT.ISRECHTS:
		    //
			// Arm staat in een uiterste stand. Eindschakelaar is ingeschakeld.
			// Zodra de arm weer wordt bewogen verandert de state.
			//
		
			GVL.Ix_OverzetterIsRechts := TRUE AND SIM.Vx_OvzIsRechtsError;	

			IF (GVL.Qx_OverzetterLinks AND NOT GVL.Qx_OverzetterRechts) THEN
				GVL.Ix_OverzetterIsRechts := FALSE;				
				Me_OvzState := OVERZETTERDUT.INHETMIDDEN;		
			END_IF			
			
		END_CASE

	END_IF	

	//
	// De status van het blokje hangt af van een aantal stuursignalen zoals waar
	// de arm zich bevindt, of er vacuum is en of er een beker lossen wordt gegeven.
	//
	
	CASE Me_BlokState OF
		OVERZETTERDUT.ISLINKS:
			//
			// Als de arm links is moet er eerste een vacuum opgebouwd worden alvorens het blokje 
			// opgepakt kan worden. Daarna verandert de state. 
			//
			
			SIM.Vx_OvzBlokGevallen 	 := INVISABLE;
			SIM.Vx_OvzBlokLinks 	 := VISABLE;
			SIM.Vx_OvzBlokOverzetter := INVISABLE;
			SIM.Vx_OvzBlokRechts 	 := INVISABLE;
			
			IF (GVL.Qx_VacuumAan AND SIM.Vx_OvzVacuumError AND GVL.Ix_OverzetterIsLinks) AND (NOT GVL.Qx_BekerLossen) THEN
				Mi_VacuumCntr := Mi_VacuumCntr + 1;
			END_IF
			
			IF (NOT GVL.Qx_VacuumAan AND SIM.Vx_OvzVacuumError) THEN
				Mi_VacuumCntr := 0;
			END_IF

			GVL.Ix_VacuumAanwezig := (Mi_VacuumCntr > 50);
	
			IF  ( GVL.Ix_VacuumAanwezig AND (Me_OvzState = OVERZETTERDUT.INHETMIDDEN)) THEN
				Me_BlokState := OVERZETTERDUT.INHETMIDDEN;
			END_IF
			
		OVERZETTERDUT.INHETMIDDEN:
			//
			// Het blokje is in beweging zolang er vacuum is. Als er geen vacuum meer is
			// valt het blokje... Indien de arm helemaal rechts is kan het blokje gelost 
			// worden. Dit moet met een Bekerlossen ondanks het feit dat er
			// geen vacuum meer is....
			//
			
			SIM.Vx_OvzBlokGevallen 	 := INVISABLE;
			SIM.Vx_OvzBlokLinks 	 := INVISABLE;
			SIM.Vx_OvzBlokOverzetter := VISABLE;
			SIM.Vx_OvzBlokRechts 	 := INVISABLE;

		 	IF (GVL.Ix_OverzetterIsRechts) AND (NOT GVL.Qx_VacuumAan) AND (GVL.Qx_BekerLossen) THEN
				GVL.Ix_VacuumAanwezig := FALSE;
				Me_BlokState := OVERZETTERDUT.ISRECHTS;		
				RETURN;		
			END_IF
			
			IF (NOT GVL.Ix_OverzetterIsRechts) AND (NOT GVL.Ix_OverzetterIsLinks) AND(NOT GVL.Qx_VacuumAan) THEN
				GVL.Ix_VacuumAanwezig := FALSE;
				Me_BlokState := OVERZETTERDUT.GEVALLEN;				
			END_IF

		OVERZETTERDUT.ISRECHTS:	
		    // 
			// Blokje is gelost. Nu is het wachten tot de overzetter terug naar links wordt gestuurd. Daarna verdwijnt
			// het blokje automatisch.
			//
			
			SIM.Vx_OvzBlokGevallen 	 := INVISABLE;
			SIM.Vx_OvzBlokLinks 	 := INVISABLE;
			SIM.Vx_OvzBlokOverzetter := INVISABLE;
			SIM.Vx_OvzBlokRechts 	 := VISABLE;
			
			IF (NOT GVL.Ix_OverzetterIsRechts) THEN
				Me_BlokState := OVERZETTERDUT.ISLINKS;					
			END_IF

		OVERZETTERDUT.GEVALLEN:
			//
			// Blokje is gevallen..... Situatie herstelt zich zodra de arm helemaal links staat.
			//
				
			SIM.Vx_OvzBlokGevallen 	 := VISABLE;
			SIM.Vx_OvzBlokLinks 	 := INVISABLE;
			SIM.Vx_OvzBlokOverzetter := INVISABLE;
			SIM.Vx_OvzBlokRechts 	 := INVISABLE;
			
			IF (GVL.Ix_OverzetterIsLinks) THEN
				Me_BlokState := OVERZETTERDUT.ISLINKS;					
			END_IF				
	END_CASE

END_PROGRAM

// Simulatie/SorterenSim
PROGRAM SorterenSim
VAR
	// Timer om sorteren te vertragen
	Fb_Pulse: BLINK;
	// Timer om sorteren te vertragen
	Fb_Trigger: F_TRIG;
	// Eerste keer om visualisatie te updaten
	Mx_FirstTime: BOOL := TRUE;
	// Afhandeling van de overzetter
	Me_SorState: SORTERENDUT := SORTERENDUT.OPDEBAND;
	// Index voor posities
	Mi_PositieIndx: INT := 1;
	// Index voor goten.
	Mi_GootIndx: INT := 1;
	// Afhandeling blokjes in goot1.
	Mb_Goot1: SorterenGootSim;
	// Afhandeling blokjes in goot2.
	Mb_Goot2: SorterenGootSim;
	// Afhandeling blokjes in goot3.
	Mb_Goot3: SorterenGootSim;
	Mx_Geplaatst: BOOL := FALSE;
	// Random nummer om kleur te bepalen
	Mi_Random: UDINT := 1;	
END_VAR
VAR CONSTANT
	// Inverse logica
	INVISABLE: BOOL := TRUE;
	// Inverse logica
	VISABLE: BOOL := FALSE;
	// Kleur rood
	RED: DWORD := 16#00FF0000;
	// Kleur wit
	WHITE: DWORD := 16#00FFFFFF;
	// Stapgrootte voor bewegingen
	STEP: INT := 4;
	// Kleur zwart
	BLACK: DWORD := 16#00000000;
	// Kleur geel
	YELLOW: DWORD := 16#00FFFF00;
	// Goot 1
	GOOT1: INT := 1;
	// Goot 2
	GOOT2: INT := 2;
	// Goot 3
	GOOT3: INT := 3;
END_VAR

// Initialisatie.

IF (Mx_FirstTime) THEN
	Me_SorState := SORTERENDUT.VOLGENDEBLOK;

	SIM.Vw_SorBlokBand  := VISABLE;
	SIM.Vw_SorKleurBand := YELLOW;
	SIM.Vi_SorBlokBandX := 0;
	SIM.Vi_SorBlokBandY := 0;
	
	FOR Mi_GootIndx := 1 TO 3 DO 
		FOR Mi_PositieIndx := 1 TO 3 DO
			SIM.Vx_SorBlokGoot[Mi_GootIndx, Mi_PositieIndx ]  := INVISABLE;
			SIM.Vw_SorKleurGoot[Mi_GootIndx, Mi_PositieIndx ] := WHITE;			
		END_FOR
	END_FOR
 
	Mx_FirstTime := FALSE;
END_IF

//
// Afhandelen van de pulse events. Hierdoor loopt de simulatie los van de 
// TASK tijd.
//
Fb_Pulse(ENABLE:=TRUE,TIMELOW:=T#50MS, TIMEHIGH:=T#50MS);
Fb_Trigger(CLK:=Fb_Pulse.OUT);


//
// Only if no emergency active, start handling the simulation.
//
IF (SIM.Ix_GotenLegen) THEN
	Mx_FirstTime := TRUE;
	SIM.Ix_GotenLegen := FALSE;
	RETURN;
END_IF


// The pulse determines the speed of the cilinder to move in
// ore move out. The cilinder is only moved if the airpressure 
// is available.
//
IF (Fb_Trigger.Q) THEN
	IF (GVL.Qx_StopperUit) THEN
		SIM.Vw_SorStopperRotate := 90;
	ELSE
		SIM.Vw_SorStopperRotate := 0;		
	END_IF
	
	IF (GVL.Qx_UitvoerGoot1Uit) THEN
		SIM.Vw_SorGoot1Rotate := 45;
	ELSE
		SIM.Vw_SorGoot1Rotate := 0;		
	END_IF	

	GVL.Ix_UitvoerGoot1IsUit := (SIM.Vw_SorGoot1Rotate > 0) AND (SIM.Vx_SorGoot1UitError);
    GVL.Ix_UitvoerGoot1IsIn  := (SIM.Vw_SorGoot1Rotate = 0) AND (SIM.Vx_SorGoot1InError);	
	
	IF (GVL.Qx_UitvoerGoot2Uit) THEN
		SIM.Vw_SorGoot2Rotate := 45;
	ELSE
		SIM.Vw_SorGoot2Rotate := 0;		
	END_IF	

	GVL.Ix_UitvoerGoot2IsUit := (SIM.Vw_SorGoot2Rotate > 0);
    GVL.Ix_UitvoerGoot2IsIn  := (SIM.Vw_SorGoot2Rotate = 0);	
	
	GVL.Ix_BekerInGoot := SIM.Vx_SorInGootError AND NOT ((SIM.Vx_SorBlokGoot[1,1] = VISABLE) OR (SIM.Vx_SorBlokGoot[2,1] = VISABLE) OR (SIM.Vx_SorBlokGoot[3,1] = VISABLE) OR ((SIM.Vi_SorBlokBandY > 30) AND (SIM.Vi_SorBlokBandY < 40)));


				
	CASE Me_SorState OF
		SORTERENDUT.VOLGENDEBLOK:
			//
			// Zet alles klaar voor een volgende blokje.
			//

			Mi_Random := DINT_TO_UDINT(TIME_TO_DINT(TIME()));
			Mi_Random := SHR((Mi_Random AND 16#000000F00), 8); 
   
			IF (Mi_Random < 5) THEN
				SIM.Vw_SorKleurBand := RED;
			ELSE IF (Mi_Random < 10) THEN
					SIM.Vw_SorKleurBand := BLACK;
				ELSE 
					SIM.Vw_SorKleurBand := YELLOW;
				END_IF
			END_IF
			
			SIM.Vw_SorBlokBand := VISABLE;
			SIM.Vi_SorBlokBandX := 0;
			SIM.Vi_SorBlokBandY := 0;
	
			Me_SorState := SORTERENDUT.OPDEBAND;
		
		SORTERENDUT.OPDEBAND:
		
			//
			// Blokje ligt op de band. Verplaats tot voor de stopper.
			//
			
			IF ((GVL.Qx_MotorAfvoerAan) AND (SIM.Vx_SorMotorAfvoerError)) THEN
				SIM.Vi_SorBlokBandX := SIM.Vi_SorBlokBandX + STEP;
			END_IF
			
			GVL.Ix_StationAfvoerVrij := (SIM.Vi_SorBlokBandX < 20);
			
			IF (SIM.Vi_SorBlokBandX > 50) THEN
				Me_SorState := SORTERENDUT.VOORSTOPPER;
			END_IF
			
		SORTERENDUT.VOORSTOPPER: 
		
			//
			// Indien de stopper uit is, dan stopt het blokje en worden
			// de kleur sensoren geactiveerd. Anders loopt het blokje gewoon door
			// naar goot 1.
			//
			
			IF ((NOT GVL.Qx_StopperUit) AND (GVL.Qx_MotorAfvoerAan) AND (SIM.Vx_SorMotorAfvoerError)) THEN
				SIM.Vi_SorBlokBandX := SIM.Vi_SorBlokBandX + STEP;	
			END_IF

			IF (GVL.Qx_StopperUit) THEN
				GVL.Ix_BekerAanwezig := TRUE;
				GVL.Ix_BekerMetaal       := (SIM.Vw_SorKleurBand = YELLOW);
				GVL.Ix_BekerReflecteerd  := (SIM.Vw_SorKleurBand = YELLOW) OR (SIM.Vw_SorKleurBand = RED);
			END_IF
			
			
			IF (SIM.Vi_SorBlokBandX > 60) THEN
				Me_SorState := SORTERENDUT.NAARGOOT1;
			END_IF		
		
		
		SORTERENDUT.NAARGOOT1:
			//
			// Voor goot 1 wordt bepaald of de stopper uit staat en het blokje dus in de goot
			// gaat. Anders loopt het blokje door naar goot 2.
			//

			GVL.Ix_BekerAanwezig := FALSE;
			
			IF ((GVL.Qx_MotorAfvoerAan) AND (SIM.Vx_SorMotorAfvoerError)) THEN
				SIM.Vi_SorBlokBandX := SIM.Vi_SorBlokBandX + STEP;
			END_IF
			
			IF ((SIM.Vi_SorBlokBandX > 130) AND (GVL.Qx_MotorAfvoerAan) AND (SIM.Vx_SorMotorAfvoerError) AND (GVL.Qx_UitvoerGoot1Uit)) THEN
				Me_SorState := SORTERENDUT.INGOOT1;
			END_IF		
	
			IF ((SIM.Vi_SorBlokBandX > 130) AND (GVL.Qx_MotorAfvoerAan) AND (SIM.Vx_SorMotorAfvoerError) AND (NOT GVL.Qx_UitvoerGoot1Uit)) THEN
				Me_SorState := SORTERENDUT.NAARGOOT2;
			END_IF	
	 
		SORTERENDUT.INGOOT1:
			//
			// Blokje valt in goot 1. Hier kunnen 3 blokjes liggen. Het  blokje van de band beweegt de goot 
			// in en aan de hand van welke blokjes er al liggen wordt het eerst volgende blokje bepaald.
			// Dit blokje wordt vervolgens getoond. Daarna is het sorteren gereed. Let op dat de goot vol
			// melding even wordt getriggered als het blokje door de sensor valt.
			//
			
			IF (SIM.Vi_SorBlokBandX < 170) THEN
				SIM.Vi_SorBlokBandX := SIM.Vi_SorBlokBandX + 2*STEP;
			END_IF
			
			SIM.Vi_SorBlokBandY := SIM.Vi_SorBlokBandY + STEP;

			
			Mb_Goot1(Px_YPos:=SIM.Vi_SorBlokBandY, Px_Goot:=GOOT1);
		
			IF (Mb_Goot1.Px_Geplaatst) THEN
				Me_SorState := SORTERENDUT.GEREED;
			END_IF
			
			IF (SIM.Vx_SorBlokGoot[GOOT1, 1] = VISABLE) THEN
				Me_SorState := SORTERENDUT.VOL;
			END_IF
			
		SORTERENDUT.NAARGOOT2: 
			//
			// Voor goot 2 wordt bepaald of de stopper uit staat en het blokje dus in de goot
			// gaat. Anders loopt het blokje door naar goot 3.
			//
		
			IF ((GVL.Qx_MotorAfvoerAan) AND (SIM.Vx_SorMotorAfvoerError)) THEN
				SIM.Vi_SorBlokBandX := SIM.Vi_SorBlokBandX + STEP;
			END_IF
			
			IF ((SIM.Vi_SorBlokBandX > 230) AND (GVL.Qx_MotorAfvoerAan) AND (SIM.Vx_SorMotorAfvoerError) AND (GVL.Qx_UitvoerGoot2Uit)) THEN
				Me_SorState := SORTERENDUT.INGOOT2;
			END_IF		
	
			IF ((SIM.Vi_SorBlokBandX > 230) AND (GVL.Qx_MotorAfvoerAan) AND (SIM.Vx_SorMotorAfvoerError) AND (NOT GVL.Qx_UitvoerGoot2Uit)) THEN
				Me_SorState := SORTERENDUT.NAARGOOT3;
			END_IF	
		
		SORTERENDUT.INGOOT2:
	
			//
			// Blokje valt in goot 2. Hier kunnen 3 blokjes liggen. Het  blokje van de band beweegt de goot 
			// in en aan de hand van welke blokjes er al liggen wordt het eerst volgende blokje bepaald.
			// Dit blokje wordt vervolgens getoond. Daarna is het sorteren gereed. Let op dat de goot vol
			// melding even wordt getriggered als het blokje door de sensor valt.
			//
			
			IF (SIM.Vi_SorBlokBandX < 270) THEN
				SIM.Vi_SorBlokBandX := SIM.Vi_SorBlokBandX + 2*STEP;
			END_IF
			
			SIM.Vi_SorBlokBandY := SIM.Vi_SorBlokBandY + STEP;
					
			Mb_Goot2(Px_YPos:=SIM.Vi_SorBlokBandY, Px_Goot:=GOOT2);
		
			IF (Mb_Goot2.Px_Geplaatst) THEN
				Me_SorState := SORTERENDUT.GEREED;
			END_IF

			IF (SIM.Vx_SorBlokGoot[GOOT2, 1] = VISABLE) THEN
				Me_SorState := SORTERENDUT.VOL;
			END_IF
		
		SORTERENDUT.NAARGOOT3: 
			//
			// Er valt niks meer te stoppen. Blokje loopt door naar goot 3.
			//
		
			IF ((GVL.Qx_MotorAfvoerAan) AND (SIM.Vx_SorMotorAfvoerError)) THEN
				SIM.Vi_SorBlokBandX := SIM.Vi_SorBlokBandX + STEP;
			END_IF
			
			IF ((SIM.Vi_SorBlokBandX > 330) AND (GVL.Qx_MotorAfvoerAan) AND (SIM.Vx_SorMotorAfvoerError)) THEN
				Me_SorState := SORTERENDUT.INGOOT3;
			END_IF		
		
		SORTERENDUT.INGOOT3:
	
			//
			// Blokje valt in goot 3. Hier kunnen 3 blokjes liggen. Het  blokje van de band beweegt de goot 
			// in en aan de hand van welke blokjes er al liggen wordt het eerst volgende blokje bepaald.
			// Dit blokje wordt vervolgens getoond. Daarna is het sorteren gereed. Let op dat de goot vol
			// melding even wordt getriggered als het blokje door de sensor valt.
			//
			
			IF (SIM.Vi_SorBlokBandX < 370) THEN
				SIM.Vi_SorBlokBandX := SIM.Vi_SorBlokBandX + 2*STEP;
			END_IF
			
			SIM.Vi_SorBlokBandY := SIM.Vi_SorBlokBandY + STEP;
			
			Mb_Goot3(Px_YPos:=SIM.Vi_SorBlokBandY, Px_Goot:=GOOT3);
		
			IF (Mb_Goot3.Px_Geplaatst) THEN
				Me_SorState := SORTERENDUT.GEREED;
			END_IF
	
			IF (SIM.Vx_SorBlokGoot[GOOT3, 1] = VISABLE) THEN
				Me_SorState := SORTERENDUT.VOL;
			END_IF
		
		SORTERENDUT.GEREED:
			SIM.Vw_SorKleurBand := WHITE;
			SIM.Vw_SorBlokBand := INVISABLE;
			SIM.Vi_SorBlokBandX := 0;
			SIM.Vi_SorBlokBandY := 0;
			
			IF (NOT GVL.Qx_MotorAfvoerAan) THEN
				Me_SorState := SORTERENDUT.VOLGENDEBLOK;
			END_IF
			
		SORTERENDUT.VOL:
			RETURN;
			
	END_CASE

END_IF

END_PROGRAM

// Simulatie/SorterenGootSim
FUNCTION_BLOCK SorterenGootSim

VAR_INPUT
	// Huidige Y positie van de blok
	Px_YPos: INT;
	// Huidge goot
	Px_Goot: INT;
END_VAR
VAR
	// Index voor posities
	Mi_PositieIndx: INT := 1;	
	// Posities van de blokjes in de goot
	Mi_Posities: ARRAY[1..6] OF INT;	
END_VAR
VAR_OUTPUT
	// Er is een positie waar het blokje terecht komt.
	Px_Geplaatst: BOOL;
END_VAR
VAR
	// Eerste keer om visualisatie te updaten
	Mx_FirstTime: BOOL := TRUE;
END_VAR
VAR CONSTANT
	// Inverse logica
	INVISABLE: BOOL := TRUE;
	// Inverse logica
	VISABLE: BOOL := FALSE;

END_VAR


//
// Initialiseer de posities van de blokjes in de goot.
//

IF (Mx_FirstTime) THEN
	Mi_Posities[1] :=  40;
	Mi_Posities[2] :=  80;
	Mi_Posities[3] := 120;
	Mi_Posities[4] := 160;
	Mi_Posities[5] := 200;
	Mi_Posities[6] := 240;	
	
	Mx_FirstTime := FALSE;
END_IF

Px_Geplaatst := FALSE;

//
// Bepaal of de huidige positie van het blokje op de band dat in de goot valt
// past bij een vaste positie in de goot. Indien dit het geval is, neem dan 
// de kleur over en toon het blokje. De goot vult zich van onder naar boven.
//

FOR Mi_PositieIndx := 3 TO 1 BY -1 DO
	IF (SIM.Vx_SorBlokGoot[Px_Goot, Mi_PositieIndx] = INVISABLE) THEN
		IF (SIM.Vi_SorBlokBandY > Mi_Posities[Mi_PositieIndx] ) THEN
			SIM.Vx_SorBlokGoot[Px_Goot, Mi_PositieIndx]  := VISABLE;
			SIM.Vw_SorKleurGoot[Px_Goot, Mi_PositieIndx] := SIM.Vw_SorKleurBand;
			
			Px_Geplaatst := TRUE;
			RETURN;
		ELSE
			RETURN;
		END_IF
	END_IF
END_FOR

END_FUNCTION_BLOCK

// Programma Structured Text/Main
// Datum : 17 december 2020, Auteur: Gerard Harkema
PROGRAM Main
VAR
	sorteerStationIO	: sorteerStationIO;
	sorteerStation 		: SorteerStationClass;
	initialized 		: BOOL := FALSE;
	sorteerStationIORef	: REFERENCE TO sorteerStationIO;
END_VAR

IF NOT initialized THEN
	// Forse Persluct aanwezig
	gvl.Ix_PersluchtAanwezig 								:= TRUE;

		// Indrukken resetknop 
	sorteerStationIO.hmi.Ix_Resetknop 					REF= Ix_Resetknop;
	// Keuzeknop staat op hand
	sorteerStationIO.hmi.Ix_Hand 						REF= gvl.Ix_Hand;
	// Keuzeknop staat op auto
	sorteerStationIO.hmi.Ix_Auto 						REF= gvl.Ix_Auto;
	// Indrukken noodstop
	sorteerStationIO.hmi.Ix_Noodstop 					REF= gvl.Ix_Noodstop;
	// Bekers magazijn zijn op

	// Indrukken startknop
	sorteerStationIO.hmi.Ix_Stopknop 					REF= gvl.Ix_Stopknop;
	// Indrukken stopknop
	sorteerStationIO.hmi.Ix_Startknop 					REF= gvl.Ix_Startknop;	
	//Perslucht is aanwezig

	// Visualisatie invisible Gele vlak
	sorteerStationIO.hmi.Qx_GeleLamp 					REF= gvl.Qx_GeleLamp;
	// Visualisatie invisible groene vlak
	sorteerStationIO.hmi.Qx_GroeneLamp 					REF= gvl.Qx_GroeneLamp;
	// Visualisatie invisible rode vlak
	sorteerStationIO.hmi.Qx_RodeLamp 					REF= gvl.Qx_RodeLamp;

	sorteerStationIO.magazijn.Ix_PersluchtAanwezig		REF= gvl.Ix_PersluchtAanwezig;
	sorteerStationIO.magazijn.Ix_MagazijnLeeg			REF= gvl.Ix_MagazijnLeeg;
	sorteerStationIO.magazijn.Ix_UitstoterBekerIn 		REF= gvl.Ix_UitstoterBekerIn;
	sorteerStationIO.magazijn.Ix_UitstoterBekerUit 		REF= gvl.Ix_UitstoterBekerUit;
	sorteerStationIO.magazijn.Qx_BekerUitstoten 		REF= gvl.Qx_BekerUitstoten;

	//Werkstuk door overzetter opgepakt
	sorteerStationIO.overzetter.Ix_VacuumAanwezig 		REF= gvl.Ix_VacuumAanwezig;
	//Overzetter haalt beker op(linker pos.)
	sorteerStationIO.overzetter.Ix_OverzetterIsLinks 	REF= gvl.Ix_OverzetterIsLinks;
	//Overzetter plaatst beker op sorteerpositie
	sorteerStationIO.overzetter.Ix_OverzetterIsRechts 	REF= gvl.Ix_OverzetterIsRechts;
	//Beker aanwezig op detectiepositie
	
		//Beker oppakken
	sorteerStationIO.overzetter.Qx_VacuumAan 			REF= gvl.Qx_VacuumAan;
	//Beker loslaten
	sorteerStationIO.overzetter.Qx_BekerLossen 			REF= gvl.Qx_BekerLossen;
	//Overzetter naar bekermagazijn
	sorteerStationIO.overzetter.Qx_OverzetterLinks		REF= gvl.Qx_OverzetterLinks;
	//Overzetter naar sorteerpositie
	sorteerStationIO.overzetter.Qx_OverzetterRechts 	REF= gvl.Qx_OverzetterRechts;

	
		//Product is naar een van de goten gegaan
	sorteerStationIO.sorteerGoot.Ix_BekerInGoot 		REF= gvl.Ix_BekerInGoot;
	//Pusher uitvoergoot 1 is in
	sorteerStationIO.sorteerGoot.Ix_UitvoerGoot1IsIn 	REF= gvl.Ix_UitvoerGoot1IsIn;
	//Pusher uitvoergoot 2 is in
	sorteerStationIO.sorteerGoot.Ix_UitvoerGoot2IsIn 	REF= gvl.Ix_UitvoerGoot2IsIn;
	//Beker afvoeren is bezig
	sorteerStationIO.sorteerGoot.Ix_StationAfvoerVrij	REF= gvl.Ix_StationAfvoerVrij;
	//Pusher uitvoergoot 1 is uit
	sorteerStationIO.sorteerGoot.Ix_UitvoerGoot1IsUit	REF= gvl.Ix_UitvoerGoot1IsUit;
	//Pusher uitvoergoot 2 is uit
	sorteerStationIO.sorteerGoot.Ix_UitvoerGoot2IsUit	REF= gvl.Ix_UitvoerGoot2IsUit;

	//Transportband aan
	sorteerStationIO.sorteerGoot.Qx_MotorAfvoerAan 		REF= gvl.Qx_MotorAfvoerAan;
	//Pusher goot 1 uit
	sorteerStationIO.sorteerGoot.Qx_UitvoerGoot1Uit 	REF= gvl.Qx_UitvoerGoot1Uit;
	//Pusher goot 2 uit
	sorteerStationIO.sorteerGoot.Qx_UitvoerGoot2Uit 	REF= gvl.Qx_UitvoerGoot2Uit;
	//Beker stoppen op band voor detectie
	sorteerStationIO.sorteerGoot.Qx_StopperUit 			REF= gvl.Qx_StopperUit;
	//Uitsorteren is bezet
	sorteerStationIO.sorteerGoot.Qx_StationBezet 		REF= gvl.Qx_StationBezet;

	//Beker aanwezig op detectiepositie
	sorteerStationIO.sorteerGoot.meetstation.Ix_BekerAanwezig 			REF= gvl.Ix_BekerAanwezig;
	//Beker is van aluminium
	sorteerStationIO.sorteerGoot.meetstation.Ix_BekerMetaal 			REF= gvl.Ix_BekerMetaal;
	//Beker reflecteert en is dus niet zwart
	sorteerStationIO.sorteerGoot.meetstation.Ix_BekerReflecteerd 		REF= gvl.Ix_BekerReflecteerd;

	sorteerStationIO.sorteerGoot.uitvoerGoot1.Ix_UitvoerGootIsIn 		REF= gvl.Ix_UitvoerGoot1IsIn;
	sorteerStationIO.sorteerGoot.uitvoerGoot1.Ix_UitvoerGootIsUit 		REF= gvl.Ix_UitvoerGoot1IsUit;
	sorteerStationIO.sorteerGoot.uitvoerGoot1.Qx_UitvoerGootUit 		REF= gvl.Qx_UitvoerGoot1Uit;
	
	sorteerStationIO.sorteerGoot.uitvoerGoot2.Ix_UitvoerGootIsIn 		REF= gvl.Ix_UitvoerGoot2IsIn;
	sorteerStationIO.sorteerGoot.uitvoerGoot2.Ix_UitvoerGootIsUit 		REF= gvl.Ix_UitvoerGoot2IsUit;
	sorteerStationIO.sorteerGoot.uitvoerGoot2.Qx_UitvoerGootUit 		REF= gvl.Qx_UitvoerGoot2Uit;
	
	sorteerStationIORef REF= sorteerStationIO;
	sorteerStation.initialize(sorteerStationIORef);

	initialized := TRUE;
END_IF

sorteerStation.cycle();

END_PROGRAM

// Programma Structured Text/SorteerStationClass
// Datum : 17 december 2020, Auteur: Gerard Harkema
FUNCTION_BLOCK SorteerStationClass
VAR
	IO				: reference to sorteerStationIO;

	// ******** Magazijn ********/
	magazijn		: MagazijnClass;
	
	// ******** Overzetter ********/
	overzetter		: OverzetterClass;
	
	// ******** Sorteergoot ********/
	sorteergoot		: SorteerGootClass;

	eState 			: sorteerStationStates := sorteerStationStates.idle;
	x_Klaar 		: BOOL := FALSE;
	x_Error 		: BOOL := FALSE;
	x_Enable 		: BOOL := FALSE;

END_VAR

// ******** Magazijn ********/
	
// ******** Overzetter ********/

// ******** Sorteergoot ********/

// Datum : 17 december 2020, Auteur: Gerard Harkema
METHOD initialize
VAR_input
	IORef						: REFERENCE TO sorteerStationIO;
END_VAR
IO REF= IORef;

// ******** Magazijn ********/
magazijn.initialize(IO.magazijn);
						
// ******** Overzetter ********/
overzetter.initialize(IO.overzetter);

// ******** Sorteergoot ********/
sorteerGoot.initialize(IO.sorteerGoot);
END_METHOD

// Datum : 17 december 2020, Auteur: Gerard Harkema
METHOD cycle
VAR

END_VAR
x_Klaar := magazijn.isKlaar() 
	   AND overzetter.isKlaar()
	   AND sorteerGoot.isKlaar();

x_Error := magazijn.isError()
	   OR overzetter.isError()
	   OR sorteerGoot.isError();
	   
	   
IF x_Error THEN
	eState := sorteerStationStates.error;
END_IF

IF IO.hmi.Ix_Startknop THEN
	x_Enable := TRUE;
//	IO.hmi.Ix_Startknop := FALSE;
END_IF
	  
IF NOT IO.hmi.Ix_Stopknop THEN
	x_Enable := FALSE;
END_IF

IF IO.hmi.Ix_ResetKnop THEN
	magazijn.reset();
	overzetter.reset();
	sorteerGoot.reset();
	x_Enable := FALSE;
	eState := sorteerStationStates.wacht_op_klaar;
END_IF

IF IO.hmi.Ix_Noodstop THEN
	magazijn.noodstop();
	overzetter.noodstop();
	sorteerGoot.noodstop();
	eState := sorteerStationStates.error;
END_IF

IO.hmi.Qx_GroeneLamp	:= NOT x_Klaar;
IO.hmi.Qx_RodeLamp 	:= x_Error;

 
CASE eState OF
	sorteerStationStates.idle:
		eState := sorteerStationStates.wacht_op_klaar;
	sorteerStationStates.wacht_op_klaar:
		IF x_Klaar THEN
			eState := sorteerStationStates.wacht_enable;
		END_IF
	sorteerStationStates.wacht_enable:
		IF magazijn.isMagazijnLeeg() OR sorteerGoot.isGootVol() THEN
			IO.hmi.Qx_GeleLamp		:= TRUE;
			eState := sorteerStationStates.service;
		ELSE
			IF x_Enable THEN
				magazijn.start();
				eState := sorteerStationStates.product_uitgifte;
			END_IF
		END_IF
	sorteerStationStates.product_uitgifte:
		IF magazijn.isKlaar() THEN
			overzetter.start();
			eState := sorteerStationStates.product_overzetten;
		END_IF
	sorteerStationStates.product_overzetten:
		IF overzetter.isKlaar() THEN
			sorteerGoot.start();
			eState := sorteerStationStates.product_sorteren;
		END_IF
	sorteerStationStates.product_sorteren:
		IF sorteerGoot.isKlaar() THEN
			eState := sorteerStationStates.wacht_enable;
		END_IF
	sorteerStationStates.service:
		IF IO.hmi.Ix_Startknop THEN
//			IO.hmi.Ix_Startknop := FALSE;
			sorteerGoot.productTellerReset();
			IO.hmi.Qx_GeleLamp		:= FALSE;
			eState := sorteerStationStates.wacht_enable;
		END_IF
END_CASE;


magazijn.cycle();
overzetter.cycle();
sorteerGoot.cycle();
END_METHOD

END_FUNCTION_BLOCK

// Programma Structured Text/MagazijnClass
// Datum : 17 december 2020, Auteur: Gerard Harkema
FUNCTION_BLOCK MagazijnClass
VAR
	IO							: REFERENCE TO magazijnIO;

	xKlaar						: BOOL := FALSE;
	eState 						: magazijnStates := magazijnStates.idle;
END_VAR

// Datum : 17 december 2020, Auteur: Gerard Harkema
METHOD initialize
VAR_INPUT

	IORef		: REFERENCE TO magazijnIO;

END_VAR
IO 			REF= IORef;

eState 		:= magazijnStates.travel_in;
END_METHOD

// Datum : 17 december 2020, Auteur: Gerard Harkema
METHOD cycle
VAR_INPUT
END_VAR

CASE eState OF
	//magazijnStates.idle:
	//magazijnStates.in:
	magazijnStates.travel_out:
		IF IO.Ix_UitstoterBekerUit THEN
			eState 			:= magazijnStates.out;	
			IO.Qx_BekerUitstoten 	:= FALSE;
		END_IF
	magazijnStates.out:
		eState 				:= magazijnStates.travel_in;	
	magazijnStates.travel_in:
		IF IO.Ix_UitstoterBekerIn THEN
			eState 			:= magazijnStates.in;
			xKlaar			:= True;	
		END_IF
	
	//magazijnStates.error:
END_CASE
END_METHOD

// Datum : 17 december 2020, Auteur: Gerard Harkema
METHOD start : BOOL
VAR_INPUT
END_VAR
IF isMagazijnLeeg() THEN
	eState 				:= magazijnStates.error;
	IO.Qx_BekerUitstoten 	:= FALSE;
	start 		:= TRUE; // Failed
	RETURN;
END_IF

IF NOT Ix_PersluchtAanwezig THEN
	eState 				:= magazijnStates.error;
	IO.Qx_BekerUitstoten 	:= FALSE;
	start 		:= TRUE; // Failed
	RETURN;
END_IF

IF NOT (eState = magazijnStates.in) THEN
	eState 				:= magazijnStates.error;
	IO.Qx_BekerUitstoten 	:= FALSE;
	start 		:= TRUE; // Failed
	RETURN;	
END_IF

xKlaar 					:= FALSE;
IO.Qx_BekerUitstoten 		:= TRUE;
eState 					:= magazijnStates.travel_out;

start 			:= FALSE; // oké
END_METHOD

// Datum : 17 december 2020, Auteur: Gerard Harkema
METHOD isMagazijnLeeg : BOOL
VAR_INPUT
END_VAR
isMagazijnLeeg := Ix_MagazijnLeeg;
END_METHOD

// Datum : 17 december 2020, Auteur: Gerard Harkema
METHOD isError : BOOL
VAR_INPUT
END_VAR
isError := (eState = magazijnStates.error);
END_METHOD

// Datum : 17 december 2020, Auteur: Gerard Harkema
METHOD reset : BOOL
VAR_INPUT
END_VAR
eState 		:= magazijnStates.travel_in;
END_METHOD

// Datum : 17 december 2020, Auteur: Gerard Harkema
METHOD isKlaar : BOOL
VAR_INPUT
END_VAR
isKlaar := xKlaar;
END_METHOD

// Datum : 17 december 2020, Auteur: Gerard Harkema
METHOD noodstop
VAR_INPUT
END_VAR
eState 				:= magazijnStates.error;
IO.Qx_BekerUitstoten 	:= FALSE;
END_METHOD

END_FUNCTION_BLOCK

// Programma Structured Text/OverzetterClass
// Datum : 17 december 2020, Auteur: Gerard Harkema
FUNCTION_BLOCK OverzetterClass
VAR
	IO							: reference to overzetterIO;

	xKlaar						: BOOL := FALSE;
	eState 						: overzetterStates := overzetterStates.idle;
	
	timer						: ton;
END_VAR

// Datum : 17 december 2020, Auteur: Gerard Harkema
METHOD initialize
VAR_INPUT
	IORef		: REFERENCE TO overzetterIO;
END_VAR

IO							REF= IORef;

IO.Qx_BekerLossen			:= FALSE;
IO.Qx_VacuumAan				:= FALSE;
IO.Qx_OverzetterLinks		:= FALSE;
IO.Qx_OverzetterRechts		:= TRUE;
eState 						:= overzetterStates.ga_naar_rechts;
END_METHOD

// Datum : 17 december 2020, Auteur: Gerard Harkema
METHOD cycle
VAR
END_VAR
CASE eState OF

//	overzetterStates.idle :
	overzetterStates.ga_naar_links:
		IF IO.Ix_OverzetterIsLinks THEN
			IO.Qx_OverzetterLinks 		:= FALSE;
			IO.Qx_VacuumAan 			:= TRUE;
			eState 					:= overzetterStates.is_links;
		END_IF;
	overzetterStates.is_links:
		IF IO.Ix_VacuumAanwezig THEN
			IO.Qx_OverzetterRechts 	:= TRUE;
			eState					:= overzetterStates.ga_naar_rechts;
	END_IF
//	overzetterStates.vaccuum_aanzetten:
	overzetterStates.ga_naar_rechts:
		IF IO.Ix_OverzetterIsRechts THEN
			IO.Qx_OverzetterRechts := FALSE;
			IO.Qx_VacuumAan 		:= FALSE;
			IO.Qx_BekerLossen 		:= TRUE;
			eState := overzetterStates.is_rechts;
		END_IF
	overzetterStates.is_rechts:
		IF NOT Ix_VacuumAanwezig THEN
			IO.Qx_BekerLossen 		:= FALSE;
			IO.Qx_OverzetterLinks 	:= TRUE;
			eState 				:= overzetterStates.ga_naar_midden;
		END_IF
//	overzetterStates.vaccuum_lossen:
	overzetterStates.ga_naar_midden:
		IF timer.Q THEN
			IO.Qx_OverzetterLinks	:= FALSE;
			eState 				:= overzetterStates.is_midden;
			xKlaar 					:= TRUE;
		END_IF
		
	//overzetterStates.is_midden:
//	overzetterStates.error:
END_CASE

timer(IN:=(estate =overzetterStates.ga_naar_midden), PT:=T#2S);
END_METHOD

// Datum : 17 december 2020, Auteur: Gerard Harkema
METHOD isError : BOOL
VAR_INPUT
END_VAR
isError := (eState = overzetterStates.error);
END_METHOD

// Datum : 17 december 2020, Auteur: Gerard Harkema
METHOD isKlaar : BOOL
VAR_INPUT
END_VAR
isKlaar := xKlaar;
END_METHOD

// Datum : 17 december 2020, Auteur: Gerard Harkema
METHOD reset
VAR_INPUT
END_VAR
IO.Qx_BekerLossen			:= FALSE;
IO.Qx_VacuumAan				:= FALSE;
IO.Qx_OverzetterLinks		:= FALSE;
IO.Qx_OverzetterRechts		:= TRUE;
eState 						:= overzetterStates.ga_naar_rechts;
END_METHOD

// Datum : 17 december 2020, Auteur: Gerard Harkema
METHOD start : BOOL
VAR_INPUT
END_VAR


IF NOT (eState = overzetterStates.is_midden) THEN
	eState 				:= overzetterStates.error;
//	IO.Qx_BekerUitstoten 	:= FALSE;
	start 	:= TRUE; // Failed
	RETURN;	
END_IF

xKlaar 					:= FALSE;
IO.Qx_OverzetterLinks 		:= TRUE;
eState 					:= overzetterStates.ga_naar_links;

start			:= FALSE; // oké
END_METHOD

// Datum : 17 december 2020, Auteur: Gerard Harkema
METHOD noodstop
VAR_INPUT
END_VAR
//Beker oppakken
IO.Qx_VacuumAan 			:=FALSE;
//Beker loslaten
IO.Qx_BekerLossen 			:=FALSE;
//Overzetter naar bekermagazijn
IO.Qx_OverzetterLinks 		:=FALSE;
//Overzetter naar sorteerpositie
IO.Qx_OverzetterRechts 	:=FALSE;

eState 				:= overzetterStates.error;
END_METHOD

END_FUNCTION_BLOCK

// Programma Structured Text/SorteerGootClass
// Datum : 17 december 2020, Auteur: Gerard Harkema
FUNCTION_BLOCK SorteerGootClass
VAR

	IO 						:REFERENCE TO 	sorteerGootIO;
	
	eState					: sorteerStates := sorteerStates.idle;

	xInitialized			: BOOL := FALSE;
	xKlaar					: BOOL := FALSE;
	
	uitvoerGoot1			: UitvoerGootClass;
	uitvoerGoot2			: UitvoerGootClass;
	
	meetstation				: MeetstationClass;
	product_type			: productType := productType.onbekend;
	
	aantal_in_goot1			: UINT := 0;
	aantal_in_goot2			: UINT := 0;
	aantal_in_goot3			: UINT := 0;
	
//	timer					: TON;

END_VAR

VAR CONSTANT
	product_type_goot1		: productType := productType.metaal_blank;
	product_type_goot2		: productType := productType.kunstof_zwart;
	product_type_goot3a		: productType := productType.kunstof_rood;
	product_type_goot3b		: productType := productType.metaal_zwart;
END_VAR

IF NOT xInitialized THEN

	xInitialized				:= TRUE;

END_IF

// Datum : 17 december 2020, Auteur: Gerard Harkema
METHOD initialize
VAR_INPUT
	IORef 							:REFERENCE TO 	sorteerGootIO;
END_VAR
IO 	REF= IORef;


meetstation.initialize(IO.meetstation);
					   
uitvoerGoot1.initialize(IO.uitvoerGoot1);

uitvoerGoot2.initialize(IO.uitvoerGoot2);
	
eState := sorteerStates.wacht_op_start;
END_METHOD

// Datum : 17 december 2020, Auteur: Gerard Harkema
METHOD cycle
VAR_INPUT
END_VAR
VAR CONSTANT
	MAX_AANTAL_IN_GOOT		: UINT := 3;
END_VAR
CASE eState OF
	sorteerStates.wacht_op_start:
		IF 	((aantal_in_goot1 >= MAX_AANTAL_IN_GOOT) OR (aantal_in_goot2 >= MAX_AANTAL_IN_GOOT) OR (aantal_in_goot3 >= MAX_AANTAL_IN_GOOT)) THEN
			eState := sorteerStates.goot_vol;
		END_IF
	sorteerStates.stopper_uit:
		IF (IO.Ix_BekerInGoot AND IO.meetstation.Ix_BekerAanwezig) THEN
			eState := sorteerStates.meten;
		END_IF
	sorteerStates.meten:
		product_type := meetstation.getProductType();
		CASE product_type OF
			product_type_goot1:
				uitvoerGoot1.gaUit();
				eState := sorteerStates.uitvoer_goot_uit;
			product_type_goot2:
				uitvoerGoot2.gaUit();
				eState := sorteerStates.uitvoer_goot_uit;
			product_type_goot3a:
				eState := sorteerStates.transporteren_naar_goot;
			product_type_goot3b:
				eState := sorteerStates.transporteren_naar_goot;
			ELSE
				eState := sorteerStates.error;
		END_CASE
		Qx_StopperUit			:= FALSE;
	sorteerStates.uitvoer_goot_uit:
		CASE product_type OF
			product_type_goot1:
				IF uitvoerGoot1.isUit() THEN
					eState := sorteerStates.transporteren_naar_goot;
				END_IF
			product_type_goot2:
				IF uitvoerGoot2.isUit() THEN
					eState := sorteerStates.transporteren_naar_goot;
				END_IF
			ELSE
				eState := sorteerStates.error;
		END_CASE
	sorteerStates.transporteren_naar_goot:
		IF NOT Ix_BekerInGoot THEN
			CASE product_type OF
				product_type_goot1:
					uitvoerGoot1.gaIn();
					aantal_in_goot1 := aantal_in_goot1 + 1;
					IO.Qx_MotorAfvoerAan := FALSE;
					eState := sorteerStates.uitvoer_goot_in;
				product_type_goot2:
					uitvoerGoot2.gaIn();
					aantal_in_goot2 := aantal_in_goot3 + 2;
					IO.Qx_MotorAfvoerAan := FALSE;
					eState := sorteerStates.uitvoer_goot_in;
				product_type_goot3a:
					aantal_in_goot3 := aantal_in_goot3 + 1;
					IO.Qx_MotorAfvoerAan := FALSE;
					eState := sorteerStates.wacht_op_start;
				product_type_goot3b:
					aantal_in_goot3 := aantal_in_goot3 + 1;
					IO.Qx_MotorAfvoerAan := FALSE;
					eState := sorteerStates.wacht_op_start;
				ELSE
					eState := sorteerStates.error;
			END_CASE
			
		END_IF
	sorteerStates.uitvoer_goot_in:
		CASE product_type OF
			product_type_goot1:
				IF uitvoerGoot1.isIn() THEN
					eState := sorteerStates.wacht_op_start;
				END_IF
			product_type_goot2:
				IF uitvoerGoot2.isIn() THEN
					eState := sorteerStates.wacht_op_start;
				END_IF
			ELSE
				eState := sorteerStates.error;
		END_CASE
	sorteerStates.reset_error:
		IF(uitvoerGoot1.isIn() AND uitvoerGoot2.isIn()) THEN
			eState := sorteerStates.wacht_op_start;
		END_IF
	sorteerStates.goot_vol:
		IF 	((aantal_in_goot1 < MAX_AANTAL_IN_GOOT) AND (aantal_in_goot2 < MAX_AANTAL_IN_GOOT) AND (aantal_in_goot3 < MAX_AANTAL_IN_GOOT)) THEN
			eState := sorteerStates.wacht_op_start;
		END_IF
//	sorteerStates.error:
END_CASE

IF eState = sorteerStates.error THEN
	//Transportband aan
	IO.Qx_MotorAfvoerAan 		:= FALSE;
	IO.Qx_StopperUit 			:= FALSE;
	//Uitsorteren is bezet
	IO.Qx_StationBezet 		:= FALSE;
END_IF


uitvoerGoot1.cycle();
uitvoerGoot2.cycle();
END_METHOD

// Datum : 17 december 2020, Auteur: Gerard Harkema
METHOD isError : BOOL
VAR_INPUT
END_VAR
isError := eState = sorteerStates.error;
END_METHOD

// Datum : 17 december 2020, Auteur: Gerard Harkema
METHOD isKlaar : BOOL
VAR_INPUT
END_VAR
isKlaar := eState = sorteerStates.wacht_op_start;
END_METHOD

// Datum : 17 december 2020, Auteur: Gerard Harkema
METHOD start : BOOL
VAR_INPUT
END_VAR
IF NOT (eState = sorteerStates.wacht_op_start) THEN
	IO.Qx_StopperUit			:= FALSE;
	IO.Qx_MotorAfvoerAan 		:= FALSE;
	eState := sorteerStates.error;
	RETURN;
END_IF
//Transportband aan
IO.Qx_StopperUit			:= TRUE;
IO.Qx_MotorAfvoerAan 		:= TRUE;
eState := sorteerStates.stopper_uit;
END_METHOD

// Datum : 17 december 2020, Auteur: Gerard Harkema
METHOD reset
VAR_INPUT
END_VAR
uitvoerGoot1.reset();
uitvoerGoot2.reset();
//Transportband aan
IO.Qx_MotorAfvoerAan 		:= FALSE;
//Beker stoppen op band voor detectie
IO.Qx_StopperUit 			:= FALSE;
//Uitsorteren is bezet
IO.Qx_StationBezet 		:= FALSE;

aantal_in_goot1			:= 0;
aantal_in_goot2			:= 0;
aantal_in_goot3			:= 0;

eState := sorteerStates.reset_error;
END_METHOD

// Datum : 17 december 2020, Auteur: Gerard Harkema
METHOD noodstop
VAR_INPUT
END_VAR
//Transportband aan
IO.Qx_MotorAfvoerAan 		:= FALSE;
IO.Qx_StopperUit 			:= FALSE;
//Uitsorteren is bezet
IO.Qx_StationBezet 		:= FALSE;

eState := sorteerStates.error;
uitvoerGoot1.noodstop();
uitvoerGoot2.noodstop();
END_METHOD

// Datum : 17 december 2020, Auteur: Gerard Harkema
METHOD isGootVol : BOOL
VAR_INPUT
END_VAR
isGootVol := eState = sorteerStates.goot_vol;
END_METHOD

// Datum : 17 december 2020, Auteur: Gerard Harkema
METHOD productTellerReset
VAR_INPUT
END_VAR
aantal_in_goot1			:= 0;
aantal_in_goot2			:= 0;
aantal_in_goot3			:= 0;
END_METHOD

END_FUNCTION_BLOCK

// Programma Structured Text/UitvoerGootClass
// Datum : 17 december 2020, Auteur: Gerard Harkema
FUNCTION_BLOCK UitvoerGootClass
VAR
	IO						: REFERENCE TO uitvoerGootIO;
	eState					: uitvoerGootStates := uitvoerGootStates.idle;
END_VAR

// Datum : 17 december 2020, Auteur: Gerard Harkema
METHOD cycle
VAR_INPUT
END_VAR
CASE eState OF
//	uitvoerGootStates.idle:
//	uitvoerGootStates.is_in:
	uitvoerGootStates.ga_in:
	IF IO.Ix_UitvoerGootIsIn THEN
		eState := uitvoerGootStates.is_in;
	END_IF

//	uitvoerGootStates.is_uit:
	uitvoerGootStates.ga_uit:
	IF IO.Ix_UitvoerGootIsUit THEN
		eState := uitvoerGootStates.is_uit;
	END_IF
//	uitvoerGootStates.error:
END_CASE
END_METHOD

// Datum : 17 december 2020, Auteur: Gerard Harkema
METHOD initialize
VAR_INPUT
	IORef			: REFERENCE TO uitvoerGootIO;

END_VAR
//Pusher uitvoergoot is in
IO 	REF=	IORef;
eState := uitvoerGootStates.ga_in;
END_METHOD

// Datum : 17 december 2020, Auteur: Gerard Harkema
METHOD isError : BOOL
VAR_INPUT
END_VAR
isError := (eState = uitvoerGootStates.error);
END_METHOD

// Datum : 17 december 2020, Auteur: Gerard Harkema
METHOD noodstop
VAR_INPUT
END_VAR
IO.Qx_UitvoerGootUit := FALSE;
eState := uitvoerGootStates.error;
END_METHOD

// Datum : 17 december 2020, Auteur: Gerard Harkema
METHOD reset
VAR_INPUT
END_VAR
IO.Qx_UitvoerGootUit := FALSE;
eState := uitvoerGootStates.ga_in;
END_METHOD

// Datum : 17 december 2020, Auteur: Gerard Harkema
METHOD gaUit
VAR_INPUT
END_VAR
IF NOT (eState = uitvoerGootStates.is_in) THEN
	eState := uitvoerGootStates.error;
	return;
END_IF

IO.Qx_UitvoerGootUit := TRUE;
eState := uitvoerGootStates.ga_uit;
END_METHOD

// Datum : 17 december 2020, Auteur: Gerard Harkema
METHOD gaIn
VAR_INPUT
END_VAR
IF NOT (eState = uitvoerGootStates.is_uit) THEN
	eState := uitvoerGootStates.error;
	return;
END_IF

IO.Qx_UitvoerGootUit := FALSE;
eState := uitvoerGootStates.ga_in;
END_METHOD

// Datum : 17 december 2020, Auteur: Gerard Harkema
METHOD isUit : BOOL
VAR_INPUT
END_VAR
isUit := (eState = uitvoerGootStates.is_uit);
END_METHOD

// Datum : 17 december 2020, Auteur: Gerard Harkema
METHOD isIn : BOOL
VAR_INPUT
END_VAR
isIn := (eState = uitvoerGootStates.is_in);
END_METHOD

END_FUNCTION_BLOCK

// Programma Structured Text/MeetstationClass
// Datum : 17 december 2020, Auteur: Gerard Harkema
FUNCTION_BLOCK MeetstationClass
VAR
	IO	: reference to meetstationIO;
END_VAR

// Datum : 17 december 2020, Auteur: Gerard Harkema
METHOD initialize
VAR_INPUT

	IORef		: reference to meetstationIO;
END_VAR
IO ref= IORef;
END_METHOD

// Datum : 17 december 2020, Auteur: Gerard Harkema
METHOD getProductType : productType
VAR_INPUT
END_VAR
IF IO.Ix_BekerAanwezig THEN
	IF IO.Ix_BekerMetaal THEN
		IF IO.Ix_BekerReflecteerd THEN
			getProductType := productType.metaal_blank;
		ELSE	
			getProductType := productType.metaal_zwart;
		END_IF
	ELSE
		IF IO.Ix_BekerReflecteerd THEN
			getProductType := productType.kunstof_rood;
		ELSE	
			getProductType := productType.metaal_zwart;
		END_IF
	END_IF
ELSE
	getProductType := productType.onbekend;	
END_IF
END_METHOD

END_FUNCTION_BLOCK

// Programma Structured Text/TestProgramms/MagazijnTest
// Datum : 17 december 2020, Auteur: Gerard Harkema
PROGRAM MagazijnTest
VAR
	xInitialaized				: BOOL := FALSE;
	
	magazijnIO					: magazijnIO;
	
	// Bekers magazijn zijn op
	Ix_MagazijnLeegRef			: REFERENCE TO BOOL;
	// Beker is uit dekselmagazijn gestoten
	Ix_UitstoterBekerInRef		: REFERENCE TO BOOL;
	// Uitstoter Beker haalt nieuwe beker op
	Ix_UitstoterBekerUitRef		: REFERENCE TO BOOL;
	// Beker uit magazijn stoten
	Qx_BekerUitstotenRef		: REFERENCE TO BOOL;
	
	magazijn: MagazijnClass;
	
END_VAR

IF NOT xInitialaized THEN

	// Forse Persluct aanwezig
	gvl.Ix_PersluchtAanwezig := TRUE;
	magazijnIO.Ix_PersluchtAanwezig		REF= gvl.Ix_PersluchtAanwezig;
	magazijnIO.Ix_MagazijnLeeg			REF= gvl.Ix_MagazijnLeeg;
	magazijnIO.Ix_UitstoterBekerIn 		REF= gvl.Ix_UitstoterBekerIn;
	magazijnIO.Ix_UitstoterBekerUit 	REF= gvl.Ix_UitstoterBekerUit;
	magazijnIO.Qx_BekerUitstoten 		REF= gvl.Qx_BekerUitstoten;

	magazijn.initialize(magazijnIO);

	xInitialaized	:= TRUE;
END_IF

IF Ix_Startknop THEN
	magazijn.start();
	Ix_Startknop := FALSE;
END_IF

IF Ix_Resetknop THEN
	magazijn.reset();
END_IF

IF Ix_Noodstop THEN
	magazijn.noodstop();
END_IF

Qx_GroeneLamp := magazijn.isKlaar();
Qx_RodeLamp := magazijn.isError();
Qx_GeleLamp := magazijn.isMagazijnLeeg();
 
magazijn.cycle();

END_PROGRAM

// Programma Structured Text/TestProgramms/OverzetterTest
// Datum : 17 december 2020, Auteur: Gerard Harkema
PROGRAM OverzetterTest
VAR
	xInitialaized				: BOOL := FALSE;

	overzetterIO				: overzetterIO;

	overzetter: OverzetterClass;
	
END_VAR

IF NOT xInitialaized THEN

	// Forse Persluct aanwezig
	gvl.Ix_PersluchtAanwezig := TRUE;
	
	//Werkstuk door overzetter opgepakt
	overzetterIO.Ix_VacuumAanwezig 		REF= gvl.Ix_VacuumAanwezig;
	//Overzetter haalt beker op(linker pos.)
	overzetterIO.Ix_OverzetterIsLinks 	REF= gvl.Ix_OverzetterIsLinks;
	//Overzetter plaatst beker op sorteerpositie
	overzetterIO.Ix_OverzetterIsRechts 	REF= gvl.Ix_OverzetterIsRechts;
	//Beker aanwezig op detectiepositie
	
		//Beker oppakken
	overzetterIO.Qx_VacuumAan 			REF= gvl.Qx_VacuumAan;
	//Beker loslaten
	overzetterIO.Qx_BekerLossen 			REF= gvl.Qx_BekerLossen;
	//Overzetter naar bekermagazijn
	overzetterIO.Qx_OverzetterLinks		REF= gvl.Qx_OverzetterLinks;
	//Overzetter naar sorteerpositie
	overzetterIO.Qx_OverzetterRechts 	REF= gvl.Qx_OverzetterRechts;

	overzetter.initialize(overzetterIO);

	xInitialaized	:= TRUE;
END_IF

IF Ix_Startknop THEN
	overzetter.start();
	Ix_Startknop := FALSE;
END_IF

IF Ix_Noodstop THEN
	overzetter.noodstop();
END_IF

IF Ix_Resetknop THEN
	overzetter.reset();
END_IF

Qx_GroeneLamp := overzetter.isKlaar();
Qx_RodeLamp := overzetter.isError();
 
overzetter.cycle();

END_PROGRAM

// Programma Structured Text/TestProgramms/SorteerTest
// Datum : 17 december 2020, Auteur: Gerard Harkema
PROGRAM SorteerTest
VAR
	xInitialaized			: BOOL := FALSE;

	sorteerGootIO			: sorteerGootIO;
	
	sorteerGoot				: SorteerGootClass;
END_VAR

IF NOT xInitialaized THEN

	// Forse Persluct aanwezig
	gvl.Ix_PersluchtAanwezig := TRUE;
	
	//Product is naar een van de goten gegaan
	sorteerGootIO.Ix_BekerInGoot 		REF= gvl.Ix_BekerInGoot;
	//Pusher uitvoergoot 1 is in
	sorteerGootIO.Ix_UitvoerGoot1IsIn 	REF= gvl.Ix_UitvoerGoot1IsIn;
	//Pusher uitvoergoot 2 is in
	sorteerGootIO.Ix_UitvoerGoot2IsIn 	REF= gvl.Ix_UitvoerGoot2IsIn;
	//Beker afvoeren is bezig
	sorteerGootIO.Ix_StationAfvoerVrij	REF= gvl.Ix_StationAfvoerVrij;
	//Pusher uitvoergoot 1 is uit
	sorteerGootIO.Ix_UitvoerGoot1IsUit	REF= gvl.Ix_UitvoerGoot1IsUit;
	//Pusher uitvoergoot 2 is uit
	sorteerGootIO.Ix_UitvoerGoot2IsUit	REF= gvl.Ix_UitvoerGoot2IsUit;

	//Transportband aan
	sorteerGootIO.Qx_MotorAfvoerAan 	REF= gvl.Qx_MotorAfvoerAan;
	//Pusher goot 1 uit
	sorteerGootIO.Qx_UitvoerGoot1Uit 	REF= gvl.Qx_UitvoerGoot1Uit;
	//Pusher goot 2 uit
	sorteerGootIO.Qx_UitvoerGoot2Uit 	REF= gvl.Qx_UitvoerGoot2Uit;
	//Beker stoppen op band voor detectie
	sorteerGootIO.Qx_StopperUit 		REF= gvl.Qx_StopperUit;
	//Uitsorteren is bezet
	sorteerGootIO.Qx_StationBezet 		REF= gvl.Qx_StationBezet;

	//Beker aanwezig op detectiepositie
	sorteerGootIO.meetstation.Ix_BekerAanwezig 		REF= gvl.Ix_BekerAanwezig;
	//Beker is van aluminium
	sorteerGootIO.meetstation.Ix_BekerMetaal 			REF= gvl.Ix_BekerMetaal;
	//Beker reflecteert en is dus niet zwart
	sorteerGootIO.meetstation.Ix_BekerReflecteerd 	REF= gvl.Ix_BekerReflecteerd;

	sorteerGootIO.uitvoerGoot1.Ix_UitvoerGootIsIn 	REF= gvl.Ix_UitvoerGoot1IsIn;
	sorteerGootIO.uitvoerGoot1.Ix_UitvoerGootIsUit 	REF= gvl.Ix_UitvoerGoot1IsUit;
	sorteerGootIO.uitvoerGoot1.Qx_UitvoerGootUit 		REF= gvl.Qx_UitvoerGoot1Uit;
	
	sorteerGootIO.uitvoerGoot2.Ix_UitvoerGootIsIn 	REF= gvl.Ix_UitvoerGoot2IsIn;
	sorteerGootIO.uitvoerGoot2.Ix_UitvoerGootIsUit 	REF= gvl.Ix_UitvoerGoot2IsUit;
	sorteerGootIO.uitvoerGoot2.Qx_UitvoerGootUit 		REF= gvl.Qx_UitvoerGoot2Uit;
	
	
	sorteerGoot.initialize(sorteerGootIO);

	xInitialaized	:= TRUE;
END_IF

IF Ix_Startknop THEN
	sorteerGoot.start();
	Ix_Startknop := FALSE;
END_IF

IF Ix_Resetknop THEN
	sorteerGoot.reset();
END_IF

IF Ix_Noodstop THEN
	sorteerGoot.noodstop();
END_IF

IF SIM.Ix_GotenLegen THEN
	sorteerGoot.productTellerReset();
END_IF

Qx_GroeneLamp := sorteerGoot.isKlaar();
Qx_RodeLamp := sorteerGoot.isError();
Qx_GeleLamp := sorteerGoot.isGootVol();
 
sorteerGoot.cycle();

END_PROGRAM

// Programma Structured Text/TestProgramms/UitvoerGootTest
// Datum : 17 december 2020, Auteur: Gerard Harkema
PROGRAM UitvoerGootTest
VAR
	xInitialaized				: BOOL := FALSE;
	
	//Pusher uitvoergoo is in
	Ix_UitvoerGootIsInRef 		: REFERENCE TO BOOL;
	//Pusher uitvoergoot is uit
	Ix_UitvoerGootIsUitRef 		: REFERENCE TO BOOL;
	//Pusher goot uit
	Qx_UitvoerGootUitRef 		: REFERENCE TO BOOL;
	
	uitvoerGootIO				: uitvoerGootIO;
	
	uitvoerGoot					: UitvoerGootClass;
	
END_VAR

IF NOT xInitialaized THEN

	// Forse Persluct aanwezig
	gvl.Ix_PersluchtAanwezig := TRUE;
	
	//Pusher uitvoergoot is in
	uitvoerGootIO.Ix_UitvoerGootIsIn 	REF= gvl.Ix_UitvoerGoot1IsIn;
	//Pusher uitvoergoot is uit
	uitvoerGootIO.Ix_UitvoerGootIsUit 	REF= gvl.Ix_UitvoerGoot1IsUit;
	//Pusher goot uit
	uitvoerGootIO.Qx_UitvoerGootUit 	REF= gvl.Qx_UitvoerGoot1Uit;
		
	uitvoerGoot.initialize(uitvoerGootIO);

	xInitialaized	:= TRUE;
	Ix_Stopknop := FALSE;
END_IF

IF Ix_Startknop THEN
	uitvoerGoot.gaUit();
	Ix_Startknop := FALSE;
END_IF

IF Ix_Stopknop THEN
	uitvoerGoot.gaIn();
	Ix_Stopknop := FALSE;
END_IF

IF Ix_Resetknop THEN
	uitvoerGoot.reset();
END_IF

IF Ix_Noodstop THEN
	uitvoerGoot.noodstop();
END_IF

Qx_GroeneLamp := uitvoerGoot.isIn();
Qx_RodeLamp := uitvoerGoot.isError();
Qx_GeleLamp := uitvoerGoot.isUit();
 
uitvoerGoot.cycle();

END_PROGRAM

// Visualisaties/SorteerStationHMI
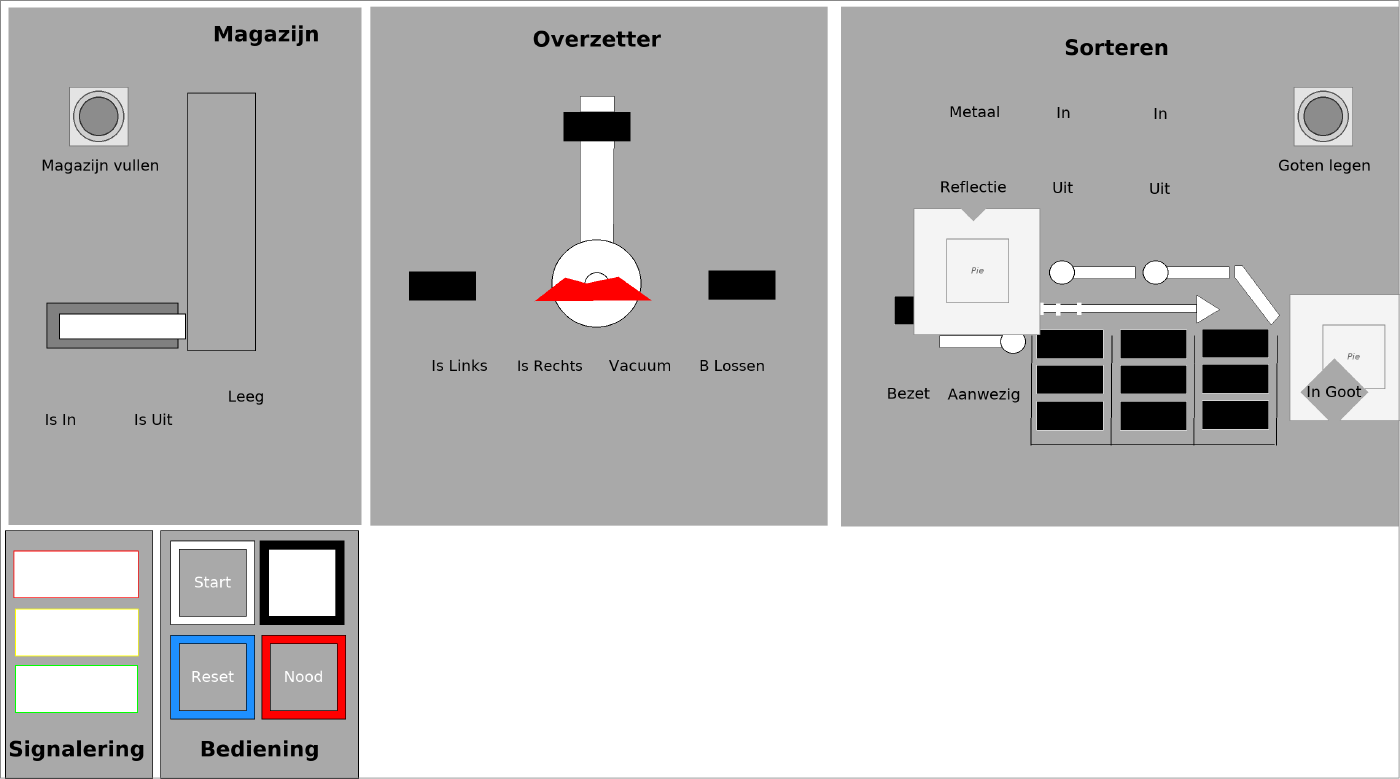
VISUALIZATION SorteerStationHMI  // 1660x924
    Rectangle (9,8 420x615)
    Polygon (247,458) (277,458) (307,458) (337,458) (292,538), "Leeg", colour toggle: Ix_MagazijnLeeg
    Polygon (72,458) (72,458) (112,498) (72,538) (32,498), "Is In", colour toggle: Ix_UitstoterBekerIn
    Polygon (182,458) (182,458) (222,498) (182,538) (142,498), "Is Uit", colour toggle: Ix_UitstoterBekerUit
    Rectangle (55,359 156x54)
    Rectangle (222,110 81x306)
    Rectangle (314,373 61x29), colour toggle: SIM.Vx_MagBlokUit
    Rectangle (227,338 61x29), colour toggle: SIM.Vx_MagBlok[2]
    Rectangle (227,302 61x29), colour toggle: SIM.Vx_MagBlok[3]
    Rectangle (227,266 61x29), colour toggle: SIM.Vx_MagBlok[4]
    Rectangle (227,373 61x29), colour toggle: SIM.Vx_MagBlok[1]
        p3560616238: SIM.Vw_MagBlok1X
    Rectangle (70,372 150x30)
        p3560616238: SIM.Vw_MagUitstoterBekerX
    Label (241,25 150x30), "Magazijn"
    Group (6,629 175x295)
        Rectangle (0,0 175x295)
        Rectangle (10,24 148x56), colour toggle: Qx_RodeLamp
        Rectangle (12,93 146x56), colour toggle: Qx_GeleLamp
        Rectangle (12,160 145x56), colour toggle: Qx_GroeneLamp
        Label (10,236 150x46), "Signalering"
    Group (190,629 235x295)
        Rectangle (0,0 235x295)
        Group (12,12 100x100)
            RoundedRectangle (0,0 100x100)
            RoundedRectangle (10,10 80x80), "Start", tooltip "Start knop", colour toggle: Ix_Startknop
                OnMouseDown: execute { Ix_Startknop := TRUE; }
                OnMouseUp: execute { Ix_Startknop := FALSE; }
        Group (118,12 100x100)
            RoundedRectangle (0,0 100x100)
            RoundedRectangle (10,10 80x80), "Stop", tooltip "Stop knop", colour toggle: Ix_Stopknop
                OnMouseDown: execute { Ix_Stopknop := FALSE; }
                OnMouseUp: execute { Ix_Stopknop := TRUE; }
        Group (12,124 100x100)
            RoundedRectangle (0,0 100x100)
            RoundedRectangle (10,10 80x80), "Reset", tooltip "Reset knop", colour toggle: Ix_Resetknop
                OnMouseDown: execute { Ix_Resetknop := TRUE; }
                OnMouseUp: execute { Ix_Resetknop := FALSE; }
        Group (120,124 100x100)
            RoundedRectangle (0,0 100x100), "Nood"
            RoundedRectangle (10,10 80x80), "Nood", tooltip "Noodstop", colour toggle: Ix_Noodstop
                OnMouseDown: execute { Ix_Noodstop := NOT Ix_Noodstop; }
        Label (43,236 150x46), "Bediening"
    Group (6,629 175x295)
        Rectangle (0,0 175x295)
        Rectangle (10,24 148x56), colour toggle: Qx_RodeLamp
        Rectangle (12,93 146x56), colour toggle: Qx_GeleLamp
        Rectangle (12,160 145x56), colour toggle: Qx_GroeneLamp
        Label (10,236 150x46), "Signalering"
    Group (190,629 235x295)
        Rectangle (0,0 235x295)
        Group (12,12 100x100)
            RoundedRectangle (0,0 100x100)
            RoundedRectangle (10,10 80x80), "Start", tooltip "Start knop", colour toggle: Ix_Startknop
                OnMouseDown: execute { Ix_Startknop := TRUE; }
                OnMouseUp: execute { Ix_Startknop := FALSE; }
        Group (118,12 100x100)
            RoundedRectangle (0,0 100x100)
            RoundedRectangle (10,10 80x80), "Stop", tooltip "Stop knop", colour toggle: Ix_Stopknop
                OnMouseDown: execute { Ix_Stopknop := FALSE; }
                OnMouseUp: execute { Ix_Stopknop := TRUE; }
        Group (12,124 100x100)
            RoundedRectangle (0,0 100x100)
            RoundedRectangle (10,10 80x80), "Reset", tooltip "Reset knop", colour toggle: Ix_Resetknop
                OnMouseDown: execute { Ix_Resetknop := TRUE; }
                OnMouseUp: execute { Ix_Resetknop := FALSE; }
        Group (120,124 100x100)
            RoundedRectangle (0,0 100x100), "Nood"
            RoundedRectangle (10,10 80x80), "Nood", tooltip "Noodstop", colour toggle: Ix_Noodstop
                OnMouseDown: execute { Ix_Noodstop := NOT Ix_Noodstop; }
        Label (43,236 150x46), "Bediening"
    Group (6,629 175x295)
        Rectangle (0,0 175x295)
        Rectangle (10,24 148x56), colour toggle: Qx_RodeLamp
        Rectangle (12,93 146x56), colour toggle: Qx_GeleLamp
        Rectangle (12,160 145x56), colour toggle: Qx_GroeneLamp
        Label (10,236 150x46), "Signalering"
    Rectangle (6,629 175x295)
    Rectangle (16,653 148x56), colour toggle: Qx_RodeLamp
    Rectangle (18,722 146x56), colour toggle: Qx_GeleLamp
    Rectangle (18,789 145x56), colour toggle: Qx_GroeneLamp
    Label (16,865 150x46), "Signalering"
    Group (190,629 235x295)
        Rectangle (0,0 235x295)
        Group (12,12 100x100)
            RoundedRectangle (0,0 100x100)
            RoundedRectangle (10,10 80x80), "Start", tooltip "Start knop", colour toggle: Ix_Startknop
                OnMouseDown: execute { Ix_Startknop := TRUE; }
                OnMouseUp: execute { Ix_Startknop := FALSE; }
        Group (118,12 100x100)
            RoundedRectangle (0,0 100x100)
            RoundedRectangle (10,10 80x80), "Stop", tooltip "Stop knop", colour toggle: Ix_Stopknop
                OnMouseDown: execute { Ix_Stopknop := FALSE; }
                OnMouseUp: execute { Ix_Stopknop := TRUE; }
        Group (12,124 100x100)
            RoundedRectangle (0,0 100x100)
            RoundedRectangle (10,10 80x80), "Reset", tooltip "Reset knop", colour toggle: Ix_Resetknop
                OnMouseDown: execute { Ix_Resetknop := TRUE; }
                OnMouseUp: execute { Ix_Resetknop := FALSE; }
        Group (120,124 100x100)
            RoundedRectangle (0,0 100x100), "Nood"
            RoundedRectangle (10,10 80x80), "Nood", tooltip "Noodstop", colour toggle: Ix_Noodstop
                OnMouseDown: execute { Ix_Noodstop := NOT Ix_Noodstop; }
        Label (43,236 150x46), "Bediening"
    Rectangle (190,629 235x295)
    Group (202,641 100x100)
        RoundedRectangle (0,0 100x100)
        RoundedRectangle (10,10 80x80), "Start", tooltip "Start knop", colour toggle: Ix_Startknop
            OnMouseDown: execute { Ix_Startknop := TRUE; }
            OnMouseUp: execute { Ix_Startknop := FALSE; }
    RoundedRectangle (202,641 100x100)
    RoundedRectangle (212,651 80x80), "Start", tooltip "Start knop", colour toggle: Ix_Startknop
        OnMouseDown: execute { Ix_Startknop := TRUE; }
        OnMouseUp: execute { Ix_Startknop := FALSE; }
    Group (308,641 100x100)
        RoundedRectangle (0,0 100x100)
        RoundedRectangle (10,10 80x80), "Stop", tooltip "Stop knop", colour toggle: Ix_Stopknop
            OnMouseDown: execute { Ix_Stopknop := FALSE; }
            OnMouseUp: execute { Ix_Stopknop := TRUE; }
    RoundedRectangle (308,641 100x100)
    RoundedRectangle (318,651 80x80), "Stop", tooltip "Stop knop", colour toggle: Ix_Stopknop
        OnMouseDown: execute { Ix_Stopknop := FALSE; }
        OnMouseUp: execute { Ix_Stopknop := TRUE; }
    Group (202,753 100x100)
        RoundedRectangle (0,0 100x100)
        RoundedRectangle (10,10 80x80), "Reset", tooltip "Reset knop", colour toggle: Ix_Resetknop
            OnMouseDown: execute { Ix_Resetknop := TRUE; }
            OnMouseUp: execute { Ix_Resetknop := FALSE; }
    RoundedRectangle (202,753 100x100)
    RoundedRectangle (212,763 80x80), "Reset", tooltip "Reset knop", colour toggle: Ix_Resetknop
        OnMouseDown: execute { Ix_Resetknop := TRUE; }
        OnMouseUp: execute { Ix_Resetknop := FALSE; }
    Group (310,753 100x100)
        RoundedRectangle (0,0 100x100), "Nood"
        RoundedRectangle (10,10 80x80), "Nood", tooltip "Noodstop", colour toggle: Ix_Noodstop
            OnMouseDown: execute { Ix_Noodstop := NOT Ix_Noodstop; }
    RoundedRectangle (310,753 100x100), "Nood"
    RoundedRectangle (320,763 80x80), "Nood", tooltip "Noodstop", colour toggle: Ix_Noodstop
        OnMouseDown: execute { Ix_Noodstop := NOT Ix_Noodstop; }
    Label (233,865 150x46), "Bediening"
    Rectangle (227,194 61x29), colour toggle: SIM.Vx_MagBlok[6]
    Rectangle (227,158 61x29), colour toggle: SIM.Vx_MagBlok[7]
    Rectangle (227,122 61x29), colour toggle: SIM.Vx_MagBlok[8]
    Rectangle (227,229 61x29), colour toggle: SIM.Vx_MagBlok[5]
    Rectangle (438,7 544x617)
    Polygon (545,394) (545,394) (585,434) (545,474) (505,434), "Is Links", colour toggle: Ix_OverzetterisLinks
    Polygon (652,394) (652,394) (692,434) (652,474) (612,434), "Is Rechts", colour toggle: Ix_OverzetterIsRechts
    Polygon (759,394) (759,394) (799,434) (759,474) (719,434), "Vacuum", colour toggle: Ix_VacuumAanwezig
    Polygon (688,131) (703,131) (728,131) (727,310) (688,310)
        p2858320360: SIM.Vx_OvzRotate
    Polygon (868,394) (868,394) (908,434) (868,474) (828,434), "B Lossen", colour toggle: Qx_BekerLossen
    Polygon (688,114) (703,114) (728,114) (728,132) (688,132), colour toggle: Qx_VacuumAan
        p2858320360: SIM.Vx_OvzRotate
    Polygon (668,133) (683,133) (747,133) (747,167) (668,167), invisible if: SIM.Vx_OvzBlokOverzetter
        p2277200375: SIM.Vx_OvzRotate
    Polygon (485,322) (500,322) (564,322) (564,356) (485,356), invisible if: SIM.Vx_OvzBlokLinks
    Polygon (840,321) (855,321) (919,321) (919,355) (840,355), invisible if: SIM.Vx_OvzBlokRechts
    Ellipse (654,284 106x104)
    Ellipse (693,323 29x27)
    Polygon (670,329) (695,336) (733,328) (772,356) (634,357), invisible if: SIM.Vx_OvzBlokGevallen
        p2277200375: SIM.Vx_OvzRotate
    Label (606,31 204x30), "Overzetter"
    Rectangle (996,7 664x618)
    Group (1197,350 249x33)
        Rectangle (0,11 222x10), colour toggle: GVL.Qx_MotorAfvoerAan
        Polygon (222,9) (222,0) (249,17) (222,33) (222,22), colour toggle: GVL.Qx_MotorAfvoerAan
        Rectangle (4,9 5x14)
        Rectangle (18,9 5x14)
        Rectangle (35,9 5x14)
        Rectangle (55,10 5x14)
        Rectangle (80,9 5x14)
    Polygon (1261,94) (1261,94) (1301,134) (1261,174) (1221,134), "In", colour toggle: GVL.Ix_UitvoerGoot1IsIn
    Polygon (1260,183) (1260,183) (1300,223) (1260,263) (1220,223), "Uit", colour toggle: GVL.Ix_UitvoerGoot1IsUit
    Polygon (1060,351) (1075,351) (1139,351) (1139,385) (1060,385), invisible if: SIM.Vw_SorBlokBand, colour variable: SIM.Vw_SorKleurBand
        p3560616238: SIM.Vi_SorBlokBandX
        p2738717112: SIM.Vi_SorBlokBandY
    Polygon (1229,391) (1244,391) (1308,391) (1308,425) (1229,425), invisible if: SIM.Vx_SorBlokGoot[1,1], colour variable: SIM.Vw_SorKleurGoot[1,1]
    Polygon (1229,433) (1244,433) (1308,433) (1308,467) (1229,467), invisible if: SIM.Vx_SorBlokGoot[1,2], colour variable: SIM.Vw_SorKleurGoot[1,2]
    Polygon (1229,476) (1244,476) (1308,476) (1308,510) (1229,510), invisible if: SIM.Vx_SorBlokGoot[1,3], colour variable: SIM.Vw_SorKleurGoot[1,3]
    Polygon (1328,391) (1343,391) (1407,391) (1407,425) (1328,425), invisible if: SIM.Vx_SorBlokGoot[2,1], colour variable: SIM.Vw_SorKleurGoot[2,1]
    Polygon (1328,433) (1343,433) (1407,433) (1407,467) (1328,467), invisible if: SIM.Vx_SorBlokGoot[2,2], colour variable: SIM.Vw_SorKleurGoot[2,2]
    Polygon (1328,476) (1343,476) (1407,476) (1407,510) (1328,510), invisible if: SIM.Vx_SorBlokGoot[2,3], colour variable: SIM.Vw_SorKleurGoot[2,3]
    Polygon (1425,390) (1440,390) (1504,390) (1504,424) (1425,424), invisible if: SIM.Vx_SorBlokGoot[3,1], colour variable: SIM.Vw_SorKleurGoot[3,1]
    Polygon (1425,432) (1440,432) (1504,432) (1504,466) (1425,466), invisible if: SIM.Vx_SorBlokGoot[3,2], colour variable: SIM.Vw_SorKleurGoot[3,2]
    Polygon (1425,475) (1440,475) (1504,475) (1504,509) (1425,509), invisible if: SIM.Vx_SorBlokGoot[3,3], colour variable: SIM.Vw_SorKleurGoot[3,3]
    Polygon (1114,398) (1169,398) (1192,398) (1192,412) (1114,412)
        p2858320360: SIM.Vw_SorStopperRotate
    Ellipse (1186,391 30x28)
    Polygon (1268,316) (1323,316) (1346,316) (1346,330) (1268,330)
        p2858320360: SIM.Vw_SorGoot1Rotate
    Ellipse (1244,309 30x28)
    Polygon (1379,316) (1434,316) (1457,316) (1457,330) (1379,330)
        p2858320360: SIM.Vw_SorGoot2Rotate
    Ellipse (1355,309 30x28)
    Polygon (1464,315) (1473,315) (1517,374) (1507,385) (1464,329)
    Group (1083,247 80x82)
        Pie (0,0 150x150)
        Pie (39,36 74x76)
    Line (1223,398) (1222,528)
    Line (1318,398) (1317,528)
    Line (1416,398) (1415,528)
    Line (1514,398) (1513,528)
    Line (1223,527) (1511,527)
    Group (1529,349 65x105)
        Pie (0,0 150x150)
        Pie (39,36 74x76)
    Polygon (1376,95) (1376,95) (1416,135) (1376,175) (1336,135), "In", colour toggle: GVL.Ix_UitvoerGoot2IsIn
    Polygon (1375,184) (1375,184) (1415,224) (1375,264) (1335,224), "Uit", colour toggle: GVL.Ix_UitvoerGoot2IsUit
    Polygon (1582,425) (1582,425) (1622,465) (1582,505) (1542,465), "In Goot", colour toggle: GVL.Ix_BekerInGoot
    Polygon (1077,427) (1077,427) (1117,467) (1077,507) (1037,467), "Bezet", colour toggle: GVL.Ix_StationAfvoerVrij
    Polygon (1156,93) (1156,93) (1196,133) (1156,173) (1116,133), "Metaal", colour toggle: GVL.Ix_BekerMetaal
    Polygon (1154,182) (1154,182) (1194,222) (1154,262) (1114,222), "Reflectie", colour toggle: GVL.Ix_BekerReflecteerd
    Polygon (1172,428) (1172,428) (1212,468) (1172,508) (1122,468), "Aanwezig", colour toggle: GVL.Ix_BekerAanwezig
    Label (1249,41 150x30), "Sorteren"
    PushSwitch (82,103 70x70), tooltip "Magazijn vullen", variable: SIM.Ix_MagazijnVullen, behaviour: TOGGLE, style: Switch-PushSwitch-Gray
    Polygon (41,184) (71,184) (101,184) (197,196) (96,212), "Magazijn vullen"
    Polygon (1493,184) (1523,184) (1553,184) (1648,198) (1548,212), "Goten legen"
    PushSwitch (1534,103 70x70), tooltip "Goten legen", variable: SIM.Ix_GotenLegen, behaviour: TOGGLE, style: Switch-PushSwitch-Gray
END_VISUALIZATION

// Visualisaties/BekerMagazijnHMI
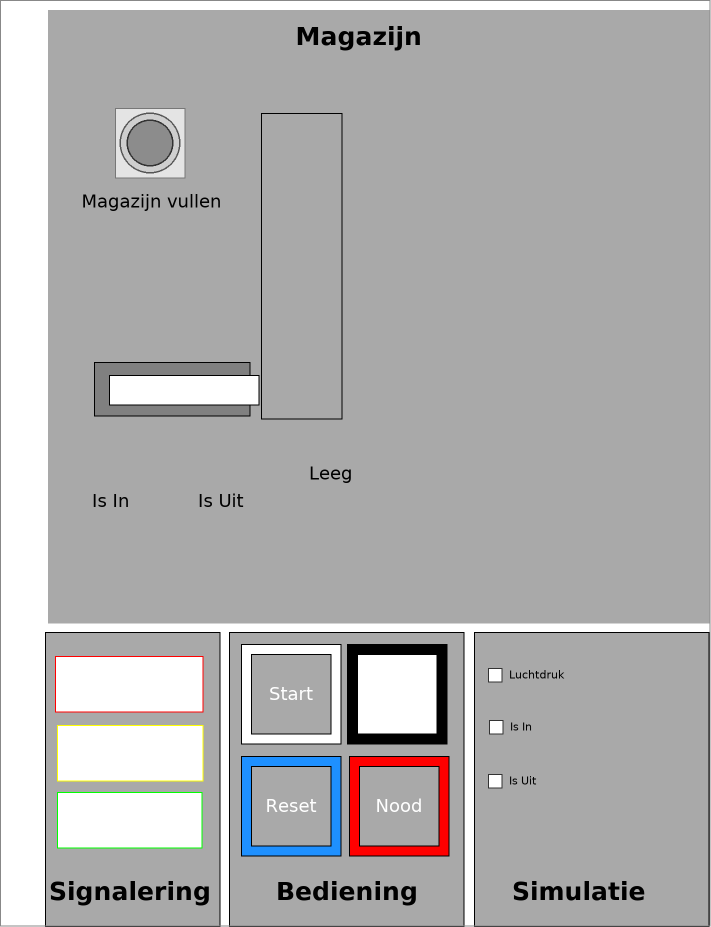
VISUALIZATION BekerMagazijnHMI  // 711x927
    Rectangle (47,9 664x615)
    Polygon (286,461) (316,461) (346,461) (376,461) (331,541), "Leeg", colour toggle: Ix_MagazijnLeeg
    Polygon (111,461) (111,461) (151,501) (111,541) (71,501), "Is In", colour toggle: Ix_UitstoterBekerIn
    Polygon (221,461) (221,461) (261,501) (221,541) (181,501), "Is Uit", colour toggle: Ix_UitstoterBekerUit
    Rectangle (94,362 156x54)
    Rectangle (261,113 81x306)
    Rectangle (353,376 61x29), colour toggle: SIM.Vx_MagBlokUit
    Rectangle (266,341 61x29), colour toggle: SIM.Vx_MagBlok[2]
    Rectangle (266,305 61x29), colour toggle: SIM.Vx_MagBlok[3]
    Rectangle (266,269 61x29), colour toggle: SIM.Vx_MagBlok[4]
    Rectangle (266,376 61x29), colour toggle: SIM.Vx_MagBlok[1]
        p3560616238: SIM.Vw_MagBlok1X
    Rectangle (109,375 150x30)
        p3560616238: SIM.Vw_MagUitstoterBekerX
    Label (284,21 150x30), "Magazijn"
    Group (45,632 664x295)
        Group (0,0 664x295)
            Group (429,0 235x295)
                Rectangle (0,0 235x295)
                Label (30,236 150x46), "Simulatie"
            Group (0,0 175x295)
                Rectangle (0,0 175x295)
                Rectangle (10,24 148x56), colour toggle: Qx_RodeLamp
                Rectangle (12,93 146x56), colour toggle: Qx_GeleLamp
                Rectangle (12,160 145x56), colour toggle: Qx_GroeneLamp
                Label (10,236 150x46), "Signalering"
            Group (184,0 235x295)
                Rectangle (0,0 235x295)
                Group (12,12 100x100)
                    RoundedRectangle (0,0 100x100)
                    RoundedRectangle (10,10 80x80), "Start", tooltip "Start knop", colour toggle: Ix_Startknop
                        OnMouseDown: execute { Ix_Startknop := TRUE; }
                        OnMouseUp: execute { Ix_Startknop := FALSE; }
                Group (118,12 100x100)
                    RoundedRectangle (0,0 100x100)
                    RoundedRectangle (10,10 80x80), "Stop", tooltip "Stop knop", colour toggle: Ix_Stopknop
                        OnMouseDown: execute { Ix_Stopknop := FALSE; }
                        OnMouseUp: execute { Ix_Stopknop := TRUE; }
                Group (12,124 100x100)
                    RoundedRectangle (0,0 100x100)
                    RoundedRectangle (10,10 80x80), "Reset", tooltip "Reset knop", colour toggle: Ix_Resetknop
                        OnMouseDown: execute { Ix_Resetknop := TRUE; }
                        OnMouseUp: execute { Ix_Resetknop := FALSE; }
                Group (120,124 100x100)
                    RoundedRectangle (0,0 100x100), "Nood"
                    RoundedRectangle (10,10 80x80), "Nood", tooltip "Noodstop", colour toggle: Ix_Noodstop
                        OnMouseDown: execute { Ix_Noodstop := NOT Ix_Noodstop; }
                Label (43,236 150x46), "Bediening"
        Checkbox (441,17 196x52), "Luchtdruk", variable: SIM.Vx_MagLuchtDrukError
        Checkbox (442,69 196x52), "Is In", variable: SIM.Vx_MagIsInError
        Checkbox (441,123 196x52), "Is Uit", variable: SIM.Vx_MagIsUitError
    Rectangle (266,197 61x29), colour toggle: SIM.Vx_MagBlok[6]
    Rectangle (266,161 61x29), colour toggle: SIM.Vx_MagBlok[7]
    Rectangle (266,125 61x29), colour toggle: SIM.Vx_MagBlok[8]
    Rectangle (266,232 61x29), colour toggle: SIM.Vx_MagBlok[5]
    Polygon (74,189) (104,189) (134,189) (229,203) (129,217), "Magazijn vullen", colour toggle: Ix_MagazijnLeeg
    PushSwitch (115,108 70x70), tooltip "Magazijn vullen", variable: SIM.Ix_MagazijnVullen, behaviour: TOGGLE, style: Switch-PushSwitch-Gray
END_VISUALIZATION

// Visualisaties/OverzetterHMI
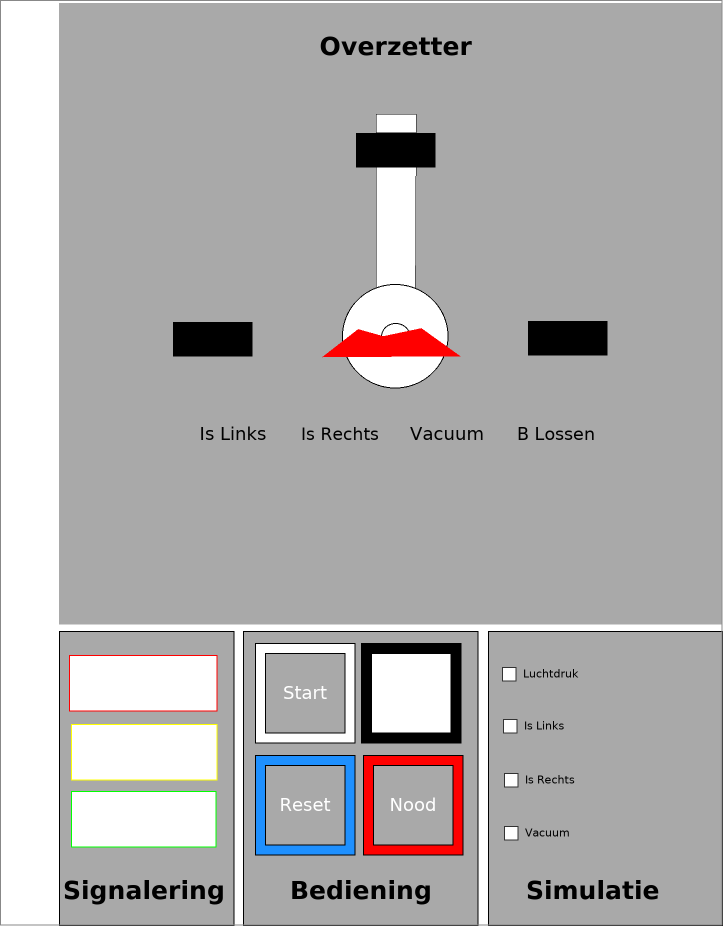
VISUALIZATION OverzetterHMI  // 723x926
    Rectangle (58,2 664x623)
    Polygon (233,394) (233,394) (273,434) (233,474) (193,434), "Is Links", colour toggle: Ix_OverzetterisLinks
    Polygon (340,394) (340,394) (380,434) (340,474) (300,434), "Is Rechts", colour toggle: Ix_OverzetterIsRechts
    Polygon (447,394) (447,394) (487,434) (447,474) (407,434), "Vacuum", colour toggle: Ix_VacuumAanwezig
    Polygon (376,131) (391,131) (416,131) (415,310) (376,310)
        p2858320360: SIM.Vx_OvzRotate
    Polygon (556,394) (556,394) (596,434) (556,474) (516,434), "B Lossen", colour toggle: Qx_BekerLossen
    Polygon (376,114) (391,114) (416,114) (416,132) (376,132), colour toggle: Qx_VacuumAan
        p2858320360: SIM.Vx_OvzRotate
    Polygon (356,133) (371,133) (435,133) (435,167) (356,167), invisible if: SIM.Vx_OvzBlokOverzetter
        p2277200375: SIM.Vx_OvzRotate
    Polygon (173,322) (188,322) (252,322) (252,356) (173,356), invisible if: SIM.Vx_OvzBlokLinks
    Polygon (528,321) (543,321) (607,321) (607,355) (528,355), invisible if: SIM.Vx_OvzBlokRechts
    Ellipse (342,284 106x104)
    Ellipse (381,323 29x27)
    Polygon (358,329) (383,336) (421,328) (460,356) (322,357), invisible if: SIM.Vx_OvzBlokGevallen
        p2277200375: SIM.Vx_OvzRotate
    Label (294,31 204x30), "Overzetter"
    Group (59,631 175x295)
        Rectangle (0,0 175x295)
        Rectangle (10,24 148x56), colour toggle: Qx_RodeLamp
        Rectangle (12,93 146x56), colour toggle: Qx_GeleLamp
        Rectangle (12,160 145x56), colour toggle: Qx_GroeneLamp
        Label (10,236 150x46), "Signalering"
    Group (243,631 235x295)
        Rectangle (0,0 235x295)
        Group (12,12 100x100)
            RoundedRectangle (0,0 100x100)
            RoundedRectangle (10,10 80x80), "Start", tooltip "Start knop", colour toggle: Ix_Startknop
                OnMouseDown: execute { Ix_Startknop := TRUE; }
                OnMouseUp: execute { Ix_Startknop := FALSE; }
        Group (118,12 100x100)
            RoundedRectangle (0,0 100x100)
            RoundedRectangle (10,10 80x80), "Stop", tooltip "Stop knop", colour toggle: Ix_Stopknop
                OnMouseDown: execute { Ix_Stopknop := FALSE; }
                OnMouseUp: execute { Ix_Stopknop := TRUE; }
        Group (12,124 100x100)
            RoundedRectangle (0,0 100x100)
            RoundedRectangle (10,10 80x80), "Reset", tooltip "Reset knop", colour toggle: Ix_Resetknop
                OnMouseDown: execute { Ix_Resetknop := TRUE; }
                OnMouseUp: execute { Ix_Resetknop := FALSE; }
        Group (120,124 100x100)
            RoundedRectangle (0,0 100x100), "Nood"
            RoundedRectangle (10,10 80x80), "Nood", tooltip "Noodstop", colour toggle: Ix_Noodstop
                OnMouseDown: execute { Ix_Noodstop := NOT Ix_Noodstop; }
        Label (43,236 150x46), "Bediening"
    Group (488,631 235x295)
        Group (0,0 235x295)
            Rectangle (0,0 235x295)
            Label (30,236 150x46), "Simulatie"
        Checkbox (12,17 196x52), "Luchtdruk", variable: SIM.Vx_OvzLuchtDrukError
        Checkbox (13,69 196x52), "Is Links", variable: SIM.Vx_OvzIsLinksError
        Checkbox (14,123 196x52), "Is Rechts", variable: SIM.Vx_OvzIsRechtsError
        Checkbox (14,176 196x52), "Vacuum", variable: SIM.Vx_OvzVacuumError
END_VISUALIZATION

